(* Offers shapes for a structuring element. *)
	{attribute 'TcIecLibraryType'}
{attribute 'Namespace' := 'Tc3_Vision'}
TYPE ETcVnStructuringElementShape : (
	TCVN_SES_RECTANGLE:=0, 	(* Rectangle *)
	TCVN_SES_CROSS:=1, 	(* Cross *)
	TCVN_SES_ELLIPSE:=2	(* Ellipse *)
) DINT;
END_TYPE

// Data Types/Enumerations/ETcVnTemplateMatchMethod

(* Offes methods for template matching. *)
	{attribute 'TcIecLibraryType'}
{attribute 'Namespace' := 'Tc3_Vision'}
TYPE ETcVnTemplateMatchMethod : (
	TCVN_TMM_SQDIFF:=0, 	(* Squared difference (supports template mask) *)
	TCVN_TMM_SQDIFF_NORMED:=1, 	(* Normalized squared difference *)
	TCVN_TMM_CCORR:=2, 	(* Cross-correlation *)
	TCVN_TMM_CCORR_NORMED:=3, 	(* Normalized cross-correlation (supports template mask) *)
	TCVN_TMM_CCOEFF:=4, 	(* Correlation coefficient *)
	TCVN_TMM_CCOEFF_NORMED:=5	(* Normalized correlation coefficient *)
) DINT;
END_TYPE

// Data Types/Enumerations/ETcVnThresholdType

(* Offers threshold types. *)
	{attribute 'TcIecLibraryType'}
{attribute 'Namespace' := 'Tc3_Vision'}
TYPE ETcVnThresholdType : (
	TCVN_TT_BINARY:=0, 	(* Binary threshold *)
	TCVN_TT_BINARY_INV:=1, 	(* Inverted binary threshold *)
	TCVN_TT_TRUNC:=2, 	(* Truncated threshold (pixels > thresh are set to thresh, others keep their value) *)
	TCVN_TT_TOZERO:=3, 	(* To zero threshold (pixels < thresh are set to zero, others keep their value) *)
	TCVN_TT_TOZERO_INV:=4, 	(* Inverted to zero threshold (pixels > thresh are set to zero, others keep their value) *)
	TCVN_TT_OTSU_BINARY:=8, 	(* Binary threshold with the threshold value selected according to the Otsu algorithm *)
	TCVN_TT_OTSU_BINARY_INV:=9, 	(* Inverted binary threshold with the threshold value selected according to the Otsu algorithm *)
	TCVN_TT_OTSU_TRUNC:=10, 	(* Truncated threshold with the threshold value selected according to the Otsu algorithm *)
	TCVN_TT_OTSU_TOZERO:=11, 	(* To zero threshold with the threshold value selected according to the Otsu algorithm *)
	TCVN_TT_OTSU_TOZERO_INV:=12, 	(* Inverted to zero threshold with the threshold value selected according to the Otsu algorithm *)
	TCVN_TT_TRIANGLE_BINARY:=16, 	(* Binary threshold with the threshold value selected according to the Triangle algorithm *)
	TCVN_TT_TRIANGLE_BINARY_INV:=17, 	(* Inverted binary threshold with the threshold value selected according to the Triangle algorithm *)
	TCVN_TT_TRIANGLE_TRUNC:=18, 	(* Truncated threshold with the threshold value selected according to the Triangle algorithm *)
	TCVN_TT_TRIANGLE_TOZERO:=19, 	(* To zero threshold with the threshold value selected according to the Triangle algorithm *)
	TCVN_TT_TRIANGLE_TOZERO_INV:=20	(* Inverted to zero threshold with the threshold value selected according to the Triangle algorithm *)
) DINT;
END_TYPE

// Data Types/Enumerations/ETcVnVectorCompareMethod

(* Offers methods for vector comparison. *)
	{attribute 'TcIecLibraryType'}
{attribute 'Namespace' := 'Tc3_Vision'}
TYPE ETcVnVectorCompareMethod : (
	TCVN_VCM_EUCLIDEAN:=0, 	(* Euclidean *)
	TCVN_VCM_ELEMENTWISE:=1	(* Elementwise *)
) DINT;
END_TYPE

// Data Types/Enumerations/ETcVnKeypointDetectionTypeAGAST

(* Offers different neighborhood types for AGAST method (For details see paper: E. Mair et al.: Adaptive and Generic Corner Detection Based on the Accelerated Segment Test, 2010). *)
	{attribute 'TcIecLibraryType'}
{attribute 'Namespace' := 'Tc3_Vision'}
TYPE ETcVnKeypointDetectionTypeAGAST : (
	TCVN_KDT_AGAST_5_8:=0, 	(* 5 of 8 *)
	TCVN_KDT_AGAST_7_12d:=1, 	(* 7 of 12 diamond *)
	TCVN_KDT_AGAST_7_12s:=2, 	(* 7 of 12 square *)
	TCVN_KDT_AGAST_9_16:=3	(* 9 of 16 *)
) DINT;
END_TYPE

// Data Types/Enumerations/ETcVnKeypointDetectionTypeFAST

(* Offers different neighborhood types for FAST method (For details see paper: E. Rosten: Machine Learning for High-speed Corner Detection, 2006). *)
	{attribute 'TcIecLibraryType'}
{attribute 'Namespace' := 'Tc3_Vision'}
TYPE ETcVnKeypointDetectionTypeFAST : (
	TCVN_KDT_FAST_5_8:=0, 	(* 5 of 8 *)
	TCVN_KDT_FAST_7_12:=1, 	(* 7 of 12 *)
	TCVN_KDT_FAST_9_16:=2	(* 9 of 16 *)
) DINT;
END_TYPE

// Data Types/Structs/TcVnParamsAGAST

(* Offers parameters for AGAST method. *)
	{attribute 'TcIecLibraryType'}
{attribute 'Namespace' := 'Tc3_Vision'}
TYPE TcVnParamsAGAST : 
	STRUCT
		(* Threshold for the intensity difference between the center pixel and its surrounding circle *)
		nThreshold : DINT := 10;
		(* If true, non-maximum suppression is applied. *)
		bNonMaxSuppression : BOOL := TRUE;
		 {attribute 'hide'}
		_reserved1 : ARRAY [1..3] OF USINT;
		(* Neighborhood type *)
		 {attribute 'GUID' := 'FA6F5C56-A2E3-4BCD-8022-41680719FF8A'}
		 {attribute 'Namespace' := 'Tc3_Vision'}
		eType : ETcVnKeypointDetectionTypeAGAST := TCVN_KDT_AGAST_9_16;
	END_STRUCT
END_TYPE

// Data Types/Structs/TcVnParamsAKAZE

(* Offers parameters for AKAZE method. *)
	{attribute 'TcIecLibraryType'}
{attribute 'Namespace' := 'Tc3_Vision'}
TYPE TcVnParamsAKAZE : 
	STRUCT
		(* Type of the descriptor *)
		 {attribute 'GUID' := 'EFB57555-E4E6-46A8-8672-7CE1494D9FAA'}
		 {attribute 'Namespace' := 'Tc3_Vision'}
		eDescrType : ETcVnFeatureDescriptorTypeAKAZE := TCVN_FDT_AKAZE_MLDB;
		(* Size of the descriptor in bits (only for MLDB; 0 = full size) *)
		nDescrSize : UDINT := 0;
		(* Number of descriptor channels (currently only 3 supported for MLDB) *)
		nDescrChannels : UDINT := 3;
		(* Detector response threshold *)
		fThreshold : REAL := 0.001;
		(* Maximum octave evolution *)
		nOctaves : UDINT := 2;
		(* Number of sublevels per scale level *)
		nOctaveLayers : UDINT := 1;
		(* Diffusivity type *)
		 {attribute 'GUID' := '808733BC-B2E0-4793-A0CE-2F414F4C0F1D'}
		 {attribute 'Namespace' := 'Tc3_Vision'}
		eDiffusivity : ETcVnDiffusivityTypeKAZE := TCVN_DT1_KAZE_PM_G2;
	END_STRUCT
END_TYPE

// Data Types/Structs/TcVnParamsBlobDetection

(* Offers parameters for blob detection *)
	{attribute 'TcIecLibraryType'}
{attribute 'Namespace' := 'Tc3_Vision'}
TYPE TcVnParamsBlobDetection : 
	STRUCT
		(* Enable filtering by area (fMinArea <= area <= fMaxArea); strongly recommended to activate for filtering noise with fMinArea. *)
		bFilterByArea : BOOL := TRUE;
		(* Enable filtering by circularity (fMinCircularity <= circularity(4pi * area / perimeter^2) <= fMaxCircularity). *)
		bFilterByCircularity : BOOL := FALSE;
		(* Enable filtering by convexity (fMinConvexity <= convexity(area / hullArea) <= fMaxConvexity). *)
		bFilterByConvexity : BOOL := FALSE;
		(* Enable filtering by eccentricity (fMinEccentricity <= eccentricity <= fMaxEccentricity). *)
		bFilterByEccentricity : BOOL := FALSE;
		(* Enable filtering by inertia ratio (fMinInertiaRatio <= inertia ratio <= fMaxInertiaRatio). *)
		bFilterByInertiaRatio : BOOL := FALSE;
		 {attribute 'hide'}
		_reserved1 : ARRAY [1..3] OF USINT;
		(* Min estimated blob area in pixel *)
		fMinArea : REAL := 10;
		(* Max estimated blob area in pixel *)
		fMaxArea : REAL := 100000000;
		(* Min circularity (1.0: ideal circle, < 1: less circular, 0: not circular at all) *)
		fMinCircularity : REAL := 0;
		(* Max circularity (1.0: ideal circle, < 1: less circular, 0: not circular at all) *)
		fMaxCircularity : REAL := 1;
		(* Min convexity (1.0: blob fully convex, < 1: less convex) *)
		fMinConvexity : REAL := 0;
		(* Max convexity (1.0: blob fully convex, < 1: less convex) *)
		fMaxConvexity : REAL := 1;
		(* Min eccentricity (0.0: circular, 1.0: linear) *)
		fMinEccentricity : REAL := 0;
		(* Max eccentricity (0.0: circular, 1.0: linear) *)
		fMaxEccentricity : REAL := 1;
		(* Min inertia ratio (1.0: equal width and height, 0.0: linear) *)
		fMinInertiaRatio : REAL := 0;
		(* Max inertia ratio (1.0: equal width and height, 0.0: linear) *)
		fMaxInertiaRatio : REAL := 1;
		(* Threshold type for internally applied threshold method (OTSU_XXX only supported for USINT images). *)
		 {attribute 'GUID' := 'C40D9A7B-C720-49F8-A5B9-1663BB6925B6'}
		 {attribute 'Namespace' := 'Tc3_Vision'}
		eThresholdType : ETcVnThresholdType := TCVN_TT_BINARY;
		(* Threshold to start with (if fThresholdStep > 0, otherwise this is the only threshold used). *)
		fMinThreshold : REAL := 30;
		(* Threshold to end with (if fThresholdStep > 0, otherwise this value is not used). *)
		fMaxThreshold : REAL := 225;
		(* Sets to 0 if only 1 threshold should be used (much faster than multiple thresholds and combining the results). *)
		fThresholdStep : REAL := 0;
		(* Minimum distance between the center points of two different blobs (only used if fThresholdStep > 0; if distance < fMinBlobDistance, the blobs are treated as the same). *)
		fMinBlobDistance : REAL := 5;
		(* Minimum number of threshold steps, for which the same contour has to be detected (only used if fThresholdStep > 0; same means center point distance < fMinBlobDistance). *)
		nMinRepeatability : UDINT := 2;
		(* Selects, which of the multi-threshold blob contours should be returned. *)
		 {attribute 'GUID' := '6B3EA399-FB72-4A3D-A347-965F9D388EB6'}
		 {attribute 'Namespace' := 'Tc3_Vision'}
		eBlobCombination : ETcVnBlobCombination := TCVN_BC_MEDIAN_THRESHOLD;
	END_STRUCT
END_TYPE

// Data Types/Structs/TcVnParamsBRISK

(* Offers parameters for BRISK method. *)
	{attribute 'TcIecLibraryType'}
{attribute 'Namespace' := 'Tc3_Vision'}
TYPE TcVnParamsBRISK : 
	STRUCT
		(* Detection threshold *)
		nThreshold : DINT := 30;
		(* Detection octaves (0 for single scale) *)
		nOctaves : UDINT := 3;
		(* Scale factor for the neighborhood pattern *)
		fPatternScale : REAL := 1;
	END_STRUCT
END_TYPE

// Data Types/Structs/TcVnParamsFAST

(* Offers parameters for FAST method. *)
	{attribute 'TcIecLibraryType'}
{attribute 'Namespace' := 'Tc3_Vision'}
TYPE TcVnParamsFAST : 
	STRUCT
		(* Threshold for the intensity difference between the center pixel and its surrounding circle *)
		nThreshold : DINT := 10;
		(* If true, non-maximum suppression is applied. *)
		bNonMaxSuppression : BOOL := TRUE;
		 {attribute 'hide'}
		_reserved1 : ARRAY [1..3] OF USINT;
		(* Neighborhood type *)
		 {attribute 'GUID' := 'FBD32F44-42B6-42E8-8896-D6A6C0F64387'}
		 {attribute 'Namespace' := 'Tc3_Vision'}
		eType : ETcVnKeypointDetectionTypeFAST := TCVN_KDT_FAST_9_16;
	END_STRUCT
END_TYPE

// Data Types/Structs/TcVnParamsGFTT

(* Offers parameters for GFTT method. *)
	{attribute 'TcIecLibraryType'}
{attribute 'Namespace' := 'Tc3_Vision'}
TYPE TcVnParamsGFTT : 
	STRUCT
		(* Maximum number of corners to return (strongest ones) *)
		nMaxCorners : UDINT := 1000;
		 {attribute 'hide'}
		_reserved1 : UDINT;
		(* Minimum accepted corner quality, relative to the strongest one *)
		fQualityLevel : LREAL := 0.01;
		(* Minimum euclidean distance between returned keypoints *)
		fMinDistance : LREAL := 1;
		(* Neighborhood block size *)
		nBlockSize : UDINT := 3;
		(* If true, a Harris detector is used instead of the default method. *)
		bUseHarrisDetector : BOOL := FALSE;
		 {attribute 'hide'}
		_reserved2 : ARRAY [1..3] OF USINT;
		(* Free parameter of the Harris detector *)
		fHarrisK : LREAL := 0.04;
	END_STRUCT
END_TYPE

// Data Types/Structs/TcVnParamsKAZE

(* Offers parameters for KAZE method *)
	{attribute 'TcIecLibraryType'}
{attribute 'Namespace' := 'Tc3_Vision'}
TYPE TcVnParamsKAZE : 
	STRUCT
		(* If true, the descriptor size is extended from the default 64 byte to 128 byte. *)
		bExtended : BOOL := FALSE;
		(* If true, upright (rotation dependent) descriptors are computed. *)
		bUpright : BOOL := FALSE;
		 {attribute 'hide'}
		_reserved1 : UINT;
		(* Detector response threshold *)
		fThreshold : REAL := 0.001;
		(* Maximum octave evolution of the image *)
		nOctaves : UDINT := 4;
		(* Number of sublevels per scale level *)
		nOctaveLayers : UDINT := 2;
		(* Diffusivity type *)
		 {attribute 'GUID' := '808733BC-B2E0-4793-A0CE-2F414F4C0F1D'}
		 {attribute 'Namespace' := 'Tc3_Vision'}
		eDiffusivity : ETcVnDiffusivityTypeKAZE := TCVN_DT1_KAZE_PM_G2;
	END_STRUCT
END_TYPE

// Data Types/Structs/TcVnParamsMSER

(* Offers parameters for MSER method *)
	{attribute 'TcIecLibraryType'}
{attribute 'Namespace' := 'Tc3_Vision'}
TYPE TcVnParamsMSER : 
	STRUCT
		(* Delta for size comparison *)
		nDelta : DINT := 5;
		(* Minimum blob size *)
		nMinArea : UDINT := 60;
		(* Maximum blob size *)
		nMaxArea : UDINT := 14400;
		 {attribute 'hide'}
		_reserved1 : UDINT;
		(* Maximum blob size variation *)
		fMaxVariation : LREAL := 0.25;
		(* Minimum MSER diversity *)
		fMinDiversity : LREAL := 0.2;
		(* Maximum evolution steps (only used for color images) *)
		nMaxEvolution : UDINT := 200;
		 {attribute 'hide'}
		_reserved2 : UDINT;
		(* Area threshold to cause re-initialization (only used for color images) *)
		fAreaThreshold : LREAL := 1.01;
		(* Minimum margin (only used for color images) *)
		fMinMargin : LREAL := 0.003;
		(* Aperture size for edge bluring (only used for color images) *)
		nEdgeBlurSize : UDINT := 5;
		 {attribute 'hide'}
		_reserved3 : UDINT;
	END_STRUCT
END_TYPE

// Data Types/Structs/TcVnParamsORB

(* Offers parameters for ORB method. *)
	{attribute 'TcIecLibraryType'}
{attribute 'Namespace' := 'Tc3_Vision'}
TYPE TcVnParamsORB : 
	STRUCT
		(* Maximum number of returned keypoints *)
		nMaxPoints : UDINT := 500;
		(* Pyramid decimation ratio (must be greater than 1, should be smaller than 2) *)
		fPyramidScale : REAL := 1.2;
		(* Number of pyramid levels *)
		nPyramidLevels : UDINT := 8;
		(* Size of the border, where no features are detected (should match nPatchSize) *)
		nEdgeThreshold : UDINT := 31;
		(* First pyramid level (currently, only 0 is supported) *)
		nFirstLevel : UDINT := 0;
		(* Number of points to produce each BRIEF descriptor element (2, 3, 4) *)
		nBriefPoints : UDINT := 2;
		(* Score type (HARRIS is more stable but slightly slower than FAST) *)
		 {attribute 'GUID' := '688ACEF5-9A4A-4447-9B39-CBC4558C02DB'}
		 {attribute 'Namespace' := 'Tc3_Vision'}
		eScoreType : ETcVnFeatureScoreTypeORB := TCVN_FST_ORB_HARRIS;
		(* Patch size of the BRIEF descriptor *)
		nPatchSize : UDINT := 31;
		(* Threshold for the FAST keypoint detection *)
		nFastThreshold : DINT := 20;
	END_STRUCT
END_TYPE

// Data Types/Structs/TcVnParamsSB

(* Offers parameters for SB method (a simple blob detector with multiple thresholds). *)
	{attribute 'TcIecLibraryType'}
{attribute 'Namespace' := 'Tc3_Vision'}
TYPE TcVnParamsSB : 
	STRUCT
		(* Enable filtering by area (fMinArea <= area < fMaxArea). *)
		bFilterByArea : BOOL := TRUE;
		(* Enable filtering by circularity (fMinCircularity <= circularity(4pi * area / perimeter^2) < fMaxCircularity). *)
		bFilterByCircularity : BOOL := FALSE;
		(* Enable filtering by color (thresholdedColor(0 or 255) = nBlobColor). *)
		bFilterByColor : BOOL := FALSE;
		(* Enable filtering by convexity (fMinConvexity <= convexity(area / hullArea) < fMaxConvexity). *)
		bFilterByConvexity : BOOL := FALSE;
		(* Enable filtering by inertia ratio (fMinInertiaRatio <= inertia ratio < fMaxInertiaRatio). *)
		bFilterByInertia : BOOL := FALSE;
		 {attribute 'hide'}
		_reserved1 : ARRAY [1..3] OF USINT;
		(* Min estimated blob area in pixel *)
		fMinArea : REAL := 25;
		(* Max estimated blob area in pixel *)
		fMaxArea : REAL := 15000;
		(* Min circularity (1.0: ideal circle, < 1: less circular, 0: not circular at all) *)
		fMinCircularity : REAL := 0;
		(* Max circularity (1.0: ideal circle, < 1: less circular, 0: not circular at all) *)
		fMaxCircularity : REAL := 1;
		(* 0 or 255 *)
		nBlobColor : USINT := 255;
		 {attribute 'hide'}
		_reserved2 : ARRAY [1..3] OF USINT;
		(* Min convexity (1.0: blob fully convex, < 1: less convex) *)
		fMinConvexity : REAL := 0;
		(* Max convexity (1.0: blob fully convex, < 1: less convex) *)
		fMaxConvexity : REAL := 1;
		(* Min inertia ratio (0.0 .. 1.0) *)
		fMinInertiaRatio : REAL := 0;
		(* Max inertia ratio (0.0 .. 1.0) *)
		fMaxInertiaRatio : REAL := 1;
		(* Min distance between different blobs *)
		fMinBlobDist : REAL := 5;
		(* Min number of same detected blobs (dist < fMinBlobDist) in different thresholds *)
		nMinRepeatability : UDINT := 2;
		(* Min threshold (start) *)
		fMinThreshold : REAL := 30;
		(* Max threshold (stop) *)
		fMaxThreshold : REAL := 225;
		(* Threshold step between min and max threshold *)
		fThresholdStep : REAL := 10;
	END_STRUCT
END_TYPE

// Version/Global_Version
{attribute 'TcGenerated'}
// This function has been automatically generated from the project information.
VAR_GLOBAL CONSTANT
	{attribute 'const_non_replaced'}
	{attribute 'linkalways'}
	stLibVersion_Tc3_Vision : ST_LibVersion := (iMajor := 4, iMinor := 0, iBuild := 2, iRevision := 13, sVersion := '4.0.2.13');
	{attribute 'const_non_replaced'}
	{attribute 'linkalways'}
	sLibraryId_Tc3_Vision : String := 'Beckhoff Automation GmbH|Tc3_Vision|4.0.2.13';
END_VAR

// Global Variables/Global_Variables

	VAR_GLOBAL
		VISION_ADS_TIMEOUT	:	TIME := TIME#5s;	(* Default ADS timeout. *)
	END_VAR

// Global Variables/TC3_VISION_IID_LIST

	VAR_GLOBAL
		IID_ITcVnColorModel	:	IID := (Data1 := 16#AFF801F3, Data2 := 16#60D0, Data3 := 16#43FA, Data4 := [16#98, 16#0F, 16#57, 16#2A, 16#62, 16#05, 16#B5, 16#AF]);	(* Interface ID for interface ITcVnColorModel *)
	END_VAR

// Function Blocks/Image Acquisition/FB_VN_GevCameraControl

	{attribute 'c++_compatible'}
	{attribute 'external_name' := 'FB_VN_GevCameraControl_GUID_B1A3978C_F082_3A85_2169_138C29DFB3DA'}
	{attribute 'TcIecLibraryType'}
	{attribute 'no_explicit_call' :='do not call this POU directly'}
	(* This FB provides the basic functionality to control a GigE Vision camera and access its calibration data. *)
	FUNCTION_BLOCK FB_VN_GevCameraControl
	VAR
		(* Internal reference to the corresponding TcVnGevImageProvider TcCOM module ID, which needs to be set via TC init symbol. *)
		{attribute 'TcInitSymbol'}
		{attribute 'TcCategoryOID' := 'TcVnGevImageProvider'}
		 {attribute 'GUID' := '18071995-0000-0000-0000-00000000000F'}
		oidITcVnGevImageProvider : OTCID;
		 {attribute 'hide'}
		_reserved1 : UINT_0_32;
		(* Internal stuff *)
		{attribute 'hide'}
		 {attribute 'GUID' := '18071995-0000-0000-0000-000000000018'}
		pInternal : PVOID;
	END_VAR


	(* Delete all images contained in the TcVnGevImageProvider TcCOM module receive queue and reset the corresponding omitted images counter. *)
	METHOD ClearImageQueue : HRESULT
END_METHOD


	(* Close the control channel to the camera. *)
	METHOD CloseCamera : HRESULT
END_METHOD


	(* Internal method *)
	{attribute 'hide'}
	METHOD FB_exit : BOOL
	VAR_INPUT
		(*  if TRUE, the exit method is called for exiting an instance that is copied afterwards (online change). *)
		bInCopyCode : BOOL;
	END_VAR
END_METHOD


	(* Internal method *)
	{attribute 'hide'}
	METHOD FB_init : BOOL
	VAR_INPUT
		(*  if TRUE, the retain variables are initialized (warm start / cold start) *)
		bInitRetains : BOOL;
		(*  if TRUE, the instance afterwards gets moved into the copy code (online change) *)
		bInCopyCode : BOOL;
	END_VAR
END_METHOD


	(* Gets the reference calibration pattern points from the TcVnGevImageProvider TcCOM module (Can be set from the calibration assistant) *)
	METHOD GetCalibPatternRef : HRESULT
	VAR_INPUT
		(* Returns the reference calibration pattern points (ContainerType_Vector_TcVnPoint3_REAL) *)
 {attribute 'GUID' := 'BC72B333-E095-465B-9693-7979773CA3B8'}
				ipCalibPatternRef : REFERENCE TO ITcVnContainer;
	END_VAR
END_METHOD


	(* Gets the camera matrix from the TcVnGevImageProvider TcCOM module (requires intrinsic calibration parameters, e.g. set by the calibration assistant) *)
	METHOD GetCameraMatrix : HRESULT
	VAR_INPUT
		(* Returns the camera matrix *)
 {attribute 'GUID' := '91A420A3-4727-4481-B3BB-170528E5BC7C'}
		 {attribute 'Namespace' := 'VN'}
				aCameraMatrix : REFERENCE TO TcVnMatrix3x3_LREAL;
	END_VAR
END_METHOD


	(* Gets the current available image (first in receive queue). *)
	METHOD GetCurrentImage : HRESULT
	VAR_INPUT
		(* Returns the image *)
 {attribute 'GUID' := '70D42C6D-6F4E-4719-8B29-2883D5D59B1C'}
				ipImage : REFERENCE TO ITcVnImage;
	END_VAR
END_METHOD


	(* Gets the current available image (first in receive queue) with undistortion applied (requires intrinsic calibration parameters in the TcVnGevImageProvider TcCOM module, e.g. set by the calibration assistant) *)
	METHOD GetCurrentImageUndistorted : HRESULT
	VAR_INPUT
		(* Returns the undistorted image *)
 {attribute 'GUID' := '70D42C6D-6F4E-4719-8B29-2883D5D59B1C'}
				ipImage : REFERENCE TO ITcVnImage;
	END_VAR
END_METHOD


	(* Gets the current available image (first in receive queue) and its corresponding GVSP info. *)
	METHOD GetCurrentImageWithGvspInfo : HRESULT
	VAR_INPUT
		(* Returns the image *)
 {attribute 'GUID' := '70D42C6D-6F4E-4719-8B29-2883D5D59B1C'}
				ipImage : REFERENCE TO ITcVnImage;
		(* Returns the GVSP info *)
 {attribute 'GUID' := '63FC7E33-91CD-44CD-9015-0BD1DC25722C'}
				stGvspInfo : REFERENCE TO GVSP_IMAGE_INFO;
	END_VAR
END_METHOD


	(* Gets the current available image (first in receive queue) with its corresponding GVSP info and undistortion applied (requires intrinsic calibration parameters in the TcVnGevImageProvider TcCOM module, e.g. set by the calibration assistant) *)
	METHOD GetCurrentImageWithGvspInfoUndistorted : HRESULT
	VAR_INPUT
		(* Returns the undistorted image *)
 {attribute 'GUID' := '70D42C6D-6F4E-4719-8B29-2883D5D59B1C'}
				ipImage : REFERENCE TO ITcVnImage;
		(* Returns the GVSP info *)
 {attribute 'GUID' := '63FC7E33-91CD-44CD-9015-0BD1DC25722C'}
				stGvspInfo : REFERENCE TO GVSP_IMAGE_INFO;
	END_VAR
END_METHOD


	(* Gets the distortion coefficients from the TcVnGevImageProvider TcCOM module (requires intrinsic calibration parameters, e.g. set by the calibration assistant) *)
	METHOD GetDistortionCoefficients : HRESULT
	VAR_INPUT
		(* Returns the distortion coefficients [k1, k2, p1, p2, k3, k4, k5, k6] *)
 {attribute 'GUID' := 'DD112102-C23A-4B37-A43A-A96400B57010'}
		 {attribute 'Namespace' := 'VN'}
				aDistortionCoefficients : REFERENCE TO TcVnArray8_LREAL;
	END_VAR
END_METHOD


	(* Gets the last received image from the queue. *)
	METHOD GetLastImageFromQueue : HRESULT
	VAR_INPUT
		(* Returns the image *)
 {attribute 'GUID' := '70D42C6D-6F4E-4719-8B29-2883D5D59B1C'}
				ipImage : REFERENCE TO ITcVnImage;
	END_VAR
END_METHOD


	(* Gets the number of omitted images since the last call of ClearImageQueue(). If the image receive queue in the TcVnGevImageProvider TcCOM module is full and a new image arrives, the first one in the queue will be deleted and the omitted counter is increased. *)
	METHOD GetOmittedImagesNum : HRESULT
	VAR_INPUT
		(* Returns the number of omitted images *)
		nOmitted : REFERENCE TO ULINT;
	END_VAR
END_METHOD


	(* Gets the rotation matrix from the TcVnGevImageProvider TcCOM module (requires extrinsic calibration parameters, e.g. set by the calibration assistant) *)
	METHOD GetRotationMatrix : HRESULT
	VAR_INPUT
		(* Returns the rotation matrix *)
 {attribute 'GUID' := '91A420A3-4727-4481-B3BB-170528E5BC7C'}
		 {attribute 'Namespace' := 'VN'}
				aRotationMatrix : REFERENCE TO TcVnMatrix3x3_LREAL;
	END_VAR
END_METHOD


	(* Gets the current state of the internal camera control state machine. *)
	METHOD GetState : ETcVnCameraState
END_METHOD


	(* Gets the translation vector from the TcVnGevImageProvider TcCOM module (requires extrinsic calibration parameters, e.g. set by the calibration assistant) *)
	METHOD GetTranslationVector : HRESULT
	VAR_INPUT
		(* Returns the translation vector *)
 {attribute 'GUID' := 'B9A67DEB-A7D1-4F25-95A3-4A82FA5C1E28'}
		 {attribute 'Namespace' := 'VN'}
				aTranslationVector : REFERENCE TO TcVnVector3_LREAL;
	END_VAR
END_METHOD


	(* Initialize the camera to the intended state (includes sending the 'InitCameraCommands' defined in the GevImageAcquisition TcCOM module to the camera). *)
	METHOD InitializeCamera : HRESULT
END_METHOD


	(* Open a control channel to the camera. *)
	METHOD OpenCamera : HRESULT
END_METHOD


	(* Reset the camera controller to initial state (might require multiple calls depending on current state, until S_OK is returned) *)
	METHOD Reset : HRESULT
END_METHOD


	(* Reset the camera features to initial state (sends the 'InitCameraCommands' defined in the GevImageAcquisition TcCOM module to the camera). *)
	METHOD ResetCameraFeatures : HRESULT
END_METHOD


	(* Sets the camera matrix to the TcVnGevImageProvider TcCOM module *)
	METHOD SetCameraMatrix : HRESULT
	VAR_INPUT
		(* The camera matrix to be copied to the TcCOM module *)
 {attribute 'GUID' := '91A420A3-4727-4481-B3BB-170528E5BC7C'}
		 {attribute 'Namespace' := 'VN'}
				aCameraMatrix : REFERENCE TO TcVnMatrix3x3_LREAL;
	END_VAR
END_METHOD


	(* Sets the distortion coefficients to the TcVnGevImageProvider TcCOM module *)
	METHOD SetDistortionCoefficients : HRESULT
	VAR_INPUT
		(* The distortion coefficients to be copied to the TcCOM module *)
 {attribute 'GUID' := 'DD112102-C23A-4B37-A43A-A96400B57010'}
		 {attribute 'Namespace' := 'VN'}
				aDistortionCoefficients : REFERENCE TO TcVnArray8_LREAL;
	END_VAR
END_METHOD


	(* Sets the rotation matrix to the TcVnGevImageProvider TcCOM module *)
	METHOD SetRotationMatrix : HRESULT
	VAR_INPUT
		(* The rotation matrix to be copied to the TcCOM module *)
 {attribute 'GUID' := '91A420A3-4727-4481-B3BB-170528E5BC7C'}
		 {attribute 'Namespace' := 'VN'}
				aRotationMatrix : REFERENCE TO TcVnMatrix3x3_LREAL;
	END_VAR
END_METHOD


	(* Sets the translation vector to the TcVnGevImageProvider TcCOM module *)
	METHOD SetTranslationVector : HRESULT
	VAR_INPUT
		(* The translation vector to be copied to the TcCOM module *)
 {attribute 'GUID' := 'B9A67DEB-A7D1-4F25-95A3-4A82FA5C1E28'}
		 {attribute 'Namespace' := 'VN'}
				aTranslationVector : REFERENCE TO TcVnVector3_LREAL;
	END_VAR
END_METHOD


	(* Send the 'StartAcquisitionCommands' defined in the TcVnGevImageProvider TcCOM module to the camera. *)
	METHOD StartAcquisition : HRESULT
END_METHOD


	(* Send the 'StopAcquisitionCommands' defined in the TcVnGevImageProvider TcCOM module to the camera. *)
	METHOD StopAcquisition : HRESULT
END_METHOD


	(* Send the 'SoftwareTriggerCommands' defined in the TcVnGevImageProvider TcCOM module to the camera. *)
	METHOD TriggerImage : HRESULT
END_METHOD

END_FUNCTION_BLOCK

// Function Blocks/Image Acquisition/FB_VN_FileSourceControl

	{attribute 'c++_compatible'}
	{attribute 'external_name' := 'FB_VN_FileSourceControl_GUID_4F53D607_3B4C_364C_3211_1EEDF57CF9AE'}
	{attribute 'TcIecLibraryType'}
	{attribute 'no_explicit_call' :='do not call this POU directly'}
	(* This FB provides access to the images send by a File Source instance. *)
	FUNCTION_BLOCK FB_VN_FileSourceControl
	VAR
		(* Internal reference to the corresponding TcVnFileImageProvider TcCOM module ID, which needs to be set via TC init symbol. *)
		{attribute 'TcInitSymbol'}
		{attribute 'TcCategoryOID' := 'TcVnFileImageProvider'}
		 {attribute 'GUID' := '18071995-0000-0000-0000-00000000000F'}
		oidITcVnFileImageProvider : OTCID;
		 {attribute 'hide'}
		_reserved1 : UINT_0_32;
		(* Internal reference to private data. *)
		{attribute 'hide'}
		 {attribute 'GUID' := '18071995-0000-0000-0000-000000000018'}
		pPriv : PVOID;
	END_VAR


	(* Internal method *)
	{attribute 'hide'}
	METHOD FB_exit : BOOL
	VAR_INPUT
		(* If TRUE, the exit method is called for exiting an instance that is copied afterwards (online change). *)
		bInCopyCode : BOOL;
	END_VAR
END_METHOD


	(* Internal method *)
	{attribute 'hide'}
	METHOD FB_init : BOOL
	VAR_INPUT
		(* If TRUE, the retain variables are initialized (warm start / cold start) *)
		bInitRetains : BOOL;
		(* If TRUE, the exit method is called for exiting an instance that is copied afterwards (online change). *)
		bInCopyCode : BOOL;
	END_VAR
END_METHOD


	(* Gets the current available image (if any). *)
	METHOD GetCurrentImage : HRESULT
	VAR_INPUT
		(* Returns the image *)
 {attribute 'GUID' := '70D42C6D-6F4E-4719-8B29-2883D5D59B1C'}
				ipImage : REFERENCE TO ITcVnImage;
	END_VAR
END_METHOD


	(* Gets the current available image (if any) and the corresponding file name. *)
	METHOD GetCurrentImageAndFileName : HRESULT
	VAR_INPUT
		(* Returns the image *)
 {attribute 'GUID' := '70D42C6D-6F4E-4719-8B29-2883D5D59B1C'}
				ipImage : REFERENCE TO ITcVnImage;
	END_VAR
	VAR_IN_OUT CONSTANT
		(* Returns the file name *)
 {attribute 'GUID' := '18071995-0000-0000-0000-00000000001A'}
				sFileName : STRING;
	END_VAR
	VAR_INPUT
		(* Define the maximum allowed length for the file name *)
		nMaxLen : UINT;
	END_VAR
END_METHOD


	(* Activates the File Source. If not in trigger mode, it will start sending images. *)
	METHOD StartAcquisition : HRESULT
END_METHOD


	(* Deactivates the File Source. It will stop sending images. *)
	METHOD StopAcquisition : HRESULT
END_METHOD


	(* Reset the controller to initial state (might require multiple calls depending on current state, until S_OK is returned) *)
	METHOD Reset : HRESULT
END_METHOD


	(* Gets the current state of the internal camera control state machine. *)
	METHOD GetState : ETcVnCameraState
END_METHOD


	(* If in trigger mode, this function triggers the next image in the list. *)
	METHOD TriggerImage : HRESULT
END_METHOD


	(* If in trigger mode, this function triggers a specific image in the list. *)
	METHOD TriggerImageExp : HRESULT
	VAR_INPUT
		(* Amount of images to skip, relative to current *)
		nSkipImages : DINT;
	END_VAR
END_METHOD


	(* If in trigger mode, this function triggers a specific image in the list by name. *)
	METHOD TriggerImageByName : HRESULT
	VAR_IN_OUT CONSTANT
		(* Name of the image to trigger *)
 {attribute 'GUID' := '18071995-0000-0000-0000-00000000001A'}
				sImageName : STRING;
	END_VAR
END_METHOD

END_FUNCTION_BLOCK

// Function Blocks/Image Acquisition/FB_VN_SimpleCameraControl

	{attribute 'c++_compatible'}
	{attribute 'external_name' := 'FB_VN_SimpleCameraControl_GUID_C57D481C_6AC1_3CDC_211F_5C11AC3CD922'}
	{attribute 'TcIecLibraryType'}
	{attribute 'no_explicit_call' :='do not call this POU directly'}
	(* This FB provides the basic functionality to control a camera or a FileSource. *)
	FUNCTION_BLOCK FB_VN_SimpleCameraControl
	VAR
		(* Internal reference to the corresponding TcVnImageProvider TcCOM module ID, which needs to be set via TC init symbol. *)
		{attribute 'TcInitSymbol'}
		{attribute 'TcCategoryOID' := 'TcVnImageProvider'}
		 {attribute 'GUID' := '18071995-0000-0000-0000-00000000000F'}
		oidITcVnImageProvider : OTCID;
		 {attribute 'hide'}
		_reserved1 : UINT_0_32;
		(* Internal stuff *)
		{attribute 'hide'}
		 {attribute 'GUID' := '18071995-0000-0000-0000-000000000018'}
		pInternal : PVOID;
	END_VAR


	(* Internal method *)
	{attribute 'hide'}
	METHOD FB_exit : BOOL
	VAR_INPUT
		(*  if TRUE, the exit method is called for exiting an instance that is copied afterwards (online change). *)
		bInCopyCode : BOOL;
	END_VAR
END_METHOD


	(* Internal method *)
	{attribute 'hide'}
	METHOD FB_init : BOOL
	VAR_INPUT
		(*  if TRUE, the retain variables are initialized (warm start / cold start) *)
		bInitRetains : BOOL;
		(*  if TRUE, the instance afterwards gets moved into the copy code (online change) *)
		bInCopyCode : BOOL;
	END_VAR
END_METHOD


	(* Get the current available image (if any). *)
	METHOD GetCurrentImage : HRESULT
	VAR_INPUT
		(* Returns the image *)
 {attribute 'GUID' := '70D42C6D-6F4E-4719-8B29-2883D5D59B1C'}
				ipImage : REFERENCE TO ITcVnImage;
	END_VAR
END_METHOD


	(* Get the current state of the internal camera control state machine. *)
	METHOD GetState : ETcVnCameraState
END_METHOD


	(* Reset the camera to initial state (might require multiple calls depending on current state, until S_OK is returned) *)
	METHOD Reset : HRESULT
END_METHOD


	(* Start the image acquisition. *)
	METHOD StartAcquisition : HRESULT
END_METHOD


	(* Stop the image acquisition. *)
	METHOD StopAcquisition : HRESULT
END_METHOD


	(* Trigger the next image. *)
	METHOD TriggerImage : HRESULT
END_METHOD

END_FUNCTION_BLOCK

// Function Blocks/File Access/FB_VN_ReadCalibrationPattern

	{attribute 'c++_compatible'}
	{attribute 'external_name' := 'FB_VN_ReadCalibrationPattern_GUID_F379CE3F_BDCE_345C_3434_ADFB5334B83F'}
	{attribute 'TcIecLibraryType'}
	(* This FB reads calibration pattern reference points from an xml file on the targte pc. *)
	FUNCTION_BLOCK FB_VN_ReadCalibrationPattern
	VAR_IN_OUT CONSTANT
		(* Full path of the file or relative path to the default directory on the target pc (%TWINCAT3DIR%\\CustomConfig\\Vision\\CalibrationPattern) *)
		 {attribute 'GUID' := '18071995-0000-0000-0000-00000000001A'}
		sFilePath : STRING;
	END_VAR
	VAR_INPUT
		(* Returns a container with the pattern points (ContainerType_Vector_TcVnPoint3_REAL) *)
		 {attribute 'GUID' := 'BC72B333-E095-465B-9693-7979773CA3B8'}
		ipDestContainer : REFERENCE TO ITcVnContainer;
		(* Reading the file is triggered by a rising edge at this input. *)
		bRead : BOOL;
	END_VAR
	VAR
		 {attribute 'hide'}
		_reserved1 : ARRAY [1..3] OF USINT;
	END_VAR
	VAR_INPUT
		(* Indicates the time before the function is cancelled. *)
		nTimeout : TIME := VISION_ADS_TIMEOUT;
	END_VAR
	VAR_OUTPUT
		(* This output remains TRUE until the function block has executed a command, but at the longest for the duration supplied to the 'nTimeout' input. While bBusy = TRUE, no new command will be accepted at the inputs. *)
		bBusy : BOOL;
		(* This output is switched to TRUE as soon as an error occurs during the execution of a command. The command-specific error code is contained in ‘nErrorId’. If the function block has a timeout error, 'bError' is TRUE and 'nErrorId' is 1861 (hexadecimal 0x745). Is reset to FALSE by the execution of a command at the inputs. *)
		bError : BOOL;
	END_VAR
	VAR
		 {attribute 'hide'}
		_reserved2 : UINT;
	END_VAR
	VAR_OUTPUT
		(* Contains the ADS error code or the command-specific error code of the last executed command. Is reset to 0 by the execution of a command at the inputs. *)
		nErrorId : UDINT;
	END_VAR
	VAR
		(* Internal parameter *)
		{attribute 'hide'}
		nAdsInvStamp : UINT;
		(* Internal parameter *)
		{attribute 'hide'}
		nAdsInvCnt : BYTE;
		(* Internal parameter *)
		{attribute 'hide'}
		ePendingRequest : BYTE;
		(* Internal parameter *)
		{attribute 'hide'}
		nTimeElapsed : TIME;
		(* Internal parameter *)
		{attribute 'hide'}
		bLastRead : BOOL;
		 {attribute 'hide'}
		_reserved3 : UINT_24_56;
		(* Internal parameter *)
		{attribute 'hide'}
		 {attribute 'GUID' := '18071995-0000-0000-0000-000000000018'}
		pBuffer : PVOID;
		(* Internal parameter *)
		{attribute 'hide'}
		 {attribute 'GUID' := '18071995-0000-0000-0000-000000000018'}
		pFilePathPending : PVOID;
	END_VAR


	(* Internal method *)
	{attribute 'hide'}
	METHOD FB_exit : BOOL
	VAR_INPUT
		(*  if TRUE, the exit method is called for exiting an instance that is copied afterwards (online change). *)
		bInCopyCode : BOOL;
	END_VAR
END_METHOD


	(* Internal method *)
	{attribute 'hide'}
	METHOD FB_init : BOOL
	VAR_INPUT
		(*  if TRUE, the retain variables are initialized (warm start / cold start) *)
		bInitRetains : BOOL;
		(*  if TRUE, the instance afterwards gets moved into the copy code (online change) *)
		bInCopyCode : BOOL;
	END_VAR
END_METHOD

END_FUNCTION_BLOCK

// Function Blocks/File Access/FB_VN_ReadContainer

	{attribute 'c++_compatible'}
	{attribute 'external_name' := 'FB_VN_ReadContainer_GUID_09A9DCF0_604B_34FA_0D21_93B42780019C'}
	{attribute 'TcIecLibraryType'}
	(* This FB reads a container from an xml file on the target pc. *)
	FUNCTION_BLOCK FB_VN_ReadContainer
	VAR_IN_OUT CONSTANT
		(* Full path of the file or relative path to the default directory on the target pc *)
		 {attribute 'GUID' := '18071995-0000-0000-0000-00000000001A'}
		sFilePath : STRING;
	END_VAR
	VAR_INPUT
		(* Returns a container with the loaded content *)
		 {attribute 'GUID' := 'BC72B333-E095-465B-9693-7979773CA3B8'}
		ipDestContainer : REFERENCE TO ITcVnContainer;
		(* The type id of the container to return. If this parameter is not set, a suitable container type will be determined automatically (except for csv files). *)
		 {attribute 'GUID' := '18071995-0000-0000-0000-000000000021'}
		nDestTypeGuid : GUID;
		(* Reading the file is triggered by a rising edge at this input. *)
		bRead : BOOL;
	END_VAR
	VAR
		 {attribute 'hide'}
		_reserved1 : ARRAY [1..3] OF USINT;
	END_VAR
	VAR_INPUT
		(* Indicates the time before the function is cancelled. *)
		nTimeout : TIME := VISION_ADS_TIMEOUT;
	END_VAR
	VAR_OUTPUT
		(* This output remains TRUE until the function block has executed a command, but at the longest for the duration supplied to the 'nTimeout' input. While bBusy = TRUE, no new command will be accepted at the inputs. *)
		bBusy : BOOL;
		(* This output is switched to TRUE as soon as an error occurs during the execution of a command. The command-specific error code is contained in ‘nErrorId’. If the function block has a timeout error, 'bError' is TRUE and 'nErrorId' is 1861 (hexadecimal 0x745). Is reset to FALSE by the execution of a command at the inputs. *)
		bError : BOOL;
	END_VAR
	VAR
		 {attribute 'hide'}
		_reserved2 : UINT;
	END_VAR
	VAR_OUTPUT
		(* Contains the ADS error code or the command-specific error code of the last executed command. Is reset to 0 by the execution of a command at the inputs. *)
		nErrorId : UDINT;
	END_VAR
	VAR
		(* Internal parameter *)
		{attribute 'hide'}
		nAdsInvStamp : UINT;
		(* Internal parameter *)
		{attribute 'hide'}
		nAdsInvCnt : BYTE;
		(* Internal parameter *)
		{attribute 'hide'}
		ePendingRequest : BYTE;
		(* Internal parameter *)
		{attribute 'hide'}
		nTimeElapsed : TIME;
		(* Internal parameter *)
		{attribute 'hide'}
		bLastRead : BOOL;
		 {attribute 'hide'}
		_reserved3 : UINT_24_56;
		(* Internal parameter *)
		{attribute 'hide'}
		 {attribute 'GUID' := '18071995-0000-0000-0000-000000000018'}
		pReadBuffer : PVOID;
		(* Internal parameter *)
		{attribute 'hide'}
		 {attribute 'GUID' := '18071995-0000-0000-0000-000000000018'}
		pWriteBuffer : PVOID;
		(* Internal parameter *)
		{attribute 'hide'}
		nWriteSize : UDINT;
		 {attribute 'hide'}
		_reserved4 : UINT_0_32;
	END_VAR


	(* Internal method *)
	{attribute 'hide'}
	METHOD FB_exit : BOOL
	VAR_INPUT
		(*  if TRUE, the exit method is called for exiting an instance that is copied afterwards (online change). *)
		bInCopyCode : BOOL;
	END_VAR
END_METHOD


	(* Internal method *)
	{attribute 'hide'}
	METHOD FB_init : BOOL
	VAR_INPUT
		(*  if TRUE, the retain variables are initialized (warm start / cold start) *)
		bInitRetains : BOOL;
		(*  if TRUE, the instance afterwards gets moved into the copy code (online change) *)
		bInCopyCode : BOOL;
	END_VAR
END_METHOD

END_FUNCTION_BLOCK

// Function Blocks/File Access/FB_VN_ReadImage

	{attribute 'c++_compatible'}
	{attribute 'external_name' := 'FB_VN_ReadImage_GUID_9CFBB651_1DA3_3417_10F1_2AF0526B92A7'}
	{attribute 'TcIecLibraryType'}
	(* This FB reads an image from a file on the target pc. *)
	FUNCTION_BLOCK FB_VN_ReadImage
	VAR_IN_OUT CONSTANT
		(* Full path of the file or relative path to the default image directory on the target pc *)
		 {attribute 'GUID' := '18071995-0000-0000-0000-00000000001A'}
		sFilePath : STRING;
	END_VAR
	VAR_INPUT
		(* Returns an image with the loaded content *)
		 {attribute 'GUID' := '70D42C6D-6F4E-4719-8B29-2883D5D59B1C'}
		ipDestImage : REFERENCE TO ITcVnImage;
		(* Reading the file is triggered by a rising edge at this input. *)
		bRead : BOOL;
	END_VAR
	VAR
		 {attribute 'hide'}
		_reserved1 : ARRAY [1..3] OF USINT;
	END_VAR
	VAR_INPUT
		(* Indicates the time before the function is cancelled. *)
		nTimeout : TIME := VISION_ADS_TIMEOUT;
	END_VAR
	VAR_OUTPUT
		(* This output remains TRUE until the function block has executed a command, but at the longest for the duration supplied to the 'nTimeout' input. While bBusy = TRUE, no new command will be accepted at the inputs. *)
		bBusy : BOOL;
		(* This output is switched to TRUE as soon as an error occurs during the execution of a command. The command-specific error code is contained in ‘nErrorId’. If the function block has a timeout error, 'bError' is TRUE and 'nErrorId' is 1861 (hexadecimal 0x745). Is reset to FALSE by the execution of a command at the inputs. *)
		bError : BOOL;
	END_VAR
	VAR
		 {attribute 'hide'}
		_reserved2 : UINT;
	END_VAR
	VAR_OUTPUT
		(* Contains the ADS error code or the command-specific error code of the last executed command. Is reset to 0 by the execution of a command at the inputs. *)
		nErrorId : UDINT;
	END_VAR
	VAR
		(* Internal parameter *)
		{attribute 'hide'}
		nAdsInvStamp : UINT;
		(* Internal parameter *)
		{attribute 'hide'}
		nAdsInvCnt : BYTE;
		(* Internal parameter *)
		{attribute 'hide'}
		ePendingRequest : BYTE;
		(* Internal parameter *)
		{attribute 'hide'}
		nTimeElapsed : TIME;
		(* Internal parameter *)
		{attribute 'hide'}
		bLastRead : BOOL;
		 {attribute 'hide'}
		_reserved3 : UINT_24_56;
		(* Internal parameter *)
		{attribute 'hide'}
		 {attribute 'GUID' := '18071995-0000-0000-0000-000000000018'}
		pBuffer : PVOID;
		(* Internal parameter *)
		{attribute 'hide'}
		 {attribute 'GUID' := '18071995-0000-0000-0000-000000000018'}
		pFilePathPending : PVOID;
	END_VAR


	(* Internal method *)
	{attribute 'hide'}
	METHOD FB_exit : BOOL
	VAR_INPUT
		(*  if TRUE, the exit method is called for exiting an instance that is copied afterwards (online change). *)
		bInCopyCode : BOOL;
	END_VAR
END_METHOD


	(* Internal method *)
	{attribute 'hide'}
	METHOD FB_init : BOOL
	VAR_INPUT
		(*  if TRUE, the retain variables are initialized (warm start / cold start) *)
		bInitRetains : BOOL;
		(*  if TRUE, the instance afterwards gets moved into the copy code (online change) *)
		bInCopyCode : BOOL;
	END_VAR
END_METHOD

END_FUNCTION_BLOCK

// Function Blocks/File Access/FB_VN_ReadMlModel

	{attribute 'c++_compatible'}
	{attribute 'external_name' := 'FB_VN_ReadMlModel_GUID_40256FBA_F075_3791_0CA2_A067683CFCA9'}
	{attribute 'TcIecLibraryType'}
	(* This FB reads a machine learning model from a file on the target pc. *)
	FUNCTION_BLOCK FB_VN_ReadMlModel
	VAR_IN_OUT CONSTANT
		(* Full path of the file or relative path to the default directory on the target pc *)
		 {attribute 'GUID' := '18071995-0000-0000-0000-00000000001A'}
		sFilePath : STRING;
	END_VAR
	VAR_INPUT
		(* Returns the loaded machine learning model *)
		 {attribute 'GUID' := 'AC23D64B-CDFA-4D43-AE8B-364A856EB3E2'}
		ipDestMlModel : REFERENCE TO ITcVnMlModel;
		(* Reading the file is triggered by a rising edge at this input. *)
		bRead : BOOL;
	END_VAR
	VAR
		 {attribute 'hide'}
		_reserved1 : ARRAY [1..3] OF USINT;
	END_VAR
	VAR_INPUT
		(* Indicates the time before the function is cancelled. *)
		nTimeout : TIME := VISION_ADS_TIMEOUT;
	END_VAR
	VAR_OUTPUT
		(* This output remains TRUE until the function block has executed a command, but at the longest for the duration supplied to the 'nTimeout' input. While bBusy = TRUE, no new command will be accepted at the inputs. *)
		bBusy : BOOL;
		(* This output is switched to TRUE as soon as an error occurs during the execution of a command. The command-specific error code is contained in ‘nErrorId’. If the function block has a timeout error, 'bError' is TRUE and 'nErrorId' is 1861 (hexadecimal 0x745). Is reset to FALSE by the execution of a command at the inputs. *)
		bError : BOOL;
	END_VAR
	VAR
		 {attribute 'hide'}
		_reserved2 : UINT;
	END_VAR
	VAR_OUTPUT
		(* Contains the ADS error code or the command-specific error code of the last executed command. Is reset to 0 by the execution of a command at the inputs. *)
		nErrorId : UDINT;
	END_VAR
	VAR
		(* Internal parameter *)
		{attribute 'hide'}
		nAdsInvStamp : UINT;
		(* Internal parameter *)
		{attribute 'hide'}
		nAdsInvCnt : BYTE;
		(* Internal parameter *)
		{attribute 'hide'}
		ePendingRequest : BYTE;
		(* Internal parameter *)
		{attribute 'hide'}
		nTimeElapsed : TIME;
		(* Internal parameter *)
		{attribute 'hide'}
		bLastRead : BOOL;
		 {attribute 'hide'}
		_reserved3 : UINT_24_56;
		(* Internal parameter *)
		{attribute 'hide'}
		 {attribute 'GUID' := '18071995-0000-0000-0000-000000000018'}
		pBuffer : PVOID;
		(* Internal parameter *)
		{attribute 'hide'}
		 {attribute 'GUID' := '18071995-0000-0000-0000-000000000018'}
		pFilePathPending : PVOID;
	END_VAR


	(* Internal method *)
	{attribute 'hide'}
	METHOD FB_exit : BOOL
	VAR_INPUT
		(*  if TRUE, the exit method is called for exiting an instance that is copied afterwards (online change). *)
		bInCopyCode : BOOL;
	END_VAR
END_METHOD


	(* Internal method *)
	{attribute 'hide'}
	METHOD FB_init : BOOL
	VAR_INPUT
		(*  if TRUE, the retain variables are initialized (warm start / cold start) *)
		bInitRetains : BOOL;
		(*  if TRUE, the instance afterwards gets moved into the copy code (online change) *)
		bInCopyCode : BOOL;
	END_VAR
END_METHOD

END_FUNCTION_BLOCK

// Function Blocks/File Access/FB_VN_WriteContainer

	{attribute 'c++_compatible'}
	{attribute 'external_name' := 'FB_VN_WriteContainer_GUID_398832D9_6000_34F8_0E2A_94AE3FB59320'}
	{attribute 'TcIecLibraryType'}
	(* This FB writes a container as an xml file to the hard drive. *)
	FUNCTION_BLOCK FB_VN_WriteContainer
	VAR_INPUT
		(* The container to write *)
		 {attribute 'GUID' := 'BC72B333-E095-465B-9693-7979773CA3B8'}
		ipContainer : REFERENCE TO ITcVnContainer;
	END_VAR
	VAR_IN_OUT CONSTANT
		(* Full path of the file or relative path to the default directory on the target pc (e.g. only a file name). If the string is empty, a file name will be generated (containing the current time). *)
		 {attribute 'GUID' := '18071995-0000-0000-0000-00000000001A'}
		sFilePath : STRING;
	END_VAR
	VAR_INPUT
		(* Container export format (default is human readable xml) *)
		 {attribute 'GUID' := 'F8305D79-70A3-4F93-A939-2FF3B8D6AF74'}
		 {attribute 'Namespace' := 'Tc3_Vision'}
		eExportFormat : ETcVnContainerExportFormat := TCVN_CEF_XML;
		(* Writing the container is triggered by a rising edge at this input. *)
		bWrite : BOOL;
	END_VAR
	VAR
		 {attribute 'hide'}
		_reserved1 : USINT;
	END_VAR
	VAR_INPUT
		(* Indicates the time before the function is cancelled. *)
		nTimeout : TIME := VISION_ADS_TIMEOUT;
	END_VAR
	VAR_OUTPUT
		(* This output remains TRUE until the function block has executed a command, but at the longest for the duration supplied to the 'nTimeout' input. While bBusy = TRUE, no new command will be accepted at the inputs. *)
		bBusy : BOOL;
		(* This output is switched to TRUE as soon as an error occurs during the execution of a command. The command-specific error code is contained in ‘nErrorId’. If the function block has a timeout error, 'bError' is TRUE and 'nErrorId' is 1861 (hexadecimal 0x745). Is reset to FALSE by the execution of a command at the inputs. *)
		bError : BOOL;
	END_VAR
	VAR
		 {attribute 'hide'}
		_reserved2 : UINT;
	END_VAR
	VAR_OUTPUT
		(* Contains the ADS error code or the command-specific error code of the last executed command. Is reset to 0 by the execution of a command at the inputs. *)
		nErrorId : UDINT;
	END_VAR
	VAR
		(* Internal parameter *)
		{attribute 'hide'}
		nAdsInvStamp : UINT;
		(* Internal parameter *)
		{attribute 'hide'}
		nAdsInvCnt : BYTE;
		 {attribute 'hide'}
		_reserved3 : USINT;
		(* Internal parameter *)
		{attribute 'hide'}
		nTimeElapsed : TIME;
		(* Internal parameter *)
		{attribute 'hide'}
		bLastWrite : BOOL;
		 {attribute 'hide'}
		_reserved4 : UINT_24_56;
	END_VAR


	(* Internal method *)
	{attribute 'hide'}
	METHOD FB_exit : BOOL
	VAR_INPUT
		(* If TRUE, the exit method is called for exiting an instance that is copied afterwards (online change). *)
		bInCopyCode : BOOL;
	END_VAR
END_METHOD


	(* Internal method *)
	{attribute 'hide'}
	METHOD FB_init : BOOL
	VAR_INPUT
		(* If TRUE, the retain variables are initialized (warm start / cold start) *)
		bInitRetains : BOOL;
		(* If TRUE, the instance afterwards gets moved into the copy code (online change) *)
		bInCopyCode : BOOL;
	END_VAR
END_METHOD

END_FUNCTION_BLOCK

// Function Blocks/File Access/FB_VN_WriteImage

	{attribute 'c++_compatible'}
	{attribute 'external_name' := 'FB_VN_WriteImage_GUID_D78879F7_FB0B_383F_0FF9_207E1DA02875'}
	{attribute 'TcIecLibraryType'}
	(* This FB writes an image to the hard drive. *)
	FUNCTION_BLOCK FB_VN_WriteImage
	VAR_INPUT
		(* The image to write *)
		 {attribute 'GUID' := '70D42C6D-6F4E-4719-8B29-2883D5D59B1C'}
		ipImage : REFERENCE TO ITcVnImage;
	END_VAR
	VAR_IN_OUT CONSTANT
		(* Full path of the file or relative path to the default directory on the target pc (e.g. only a file name). If the string is empty, a file name will be generated (containing the current time). *)
		 {attribute 'GUID' := '18071995-0000-0000-0000-00000000001A'}
		sFilePath : STRING;
	END_VAR
	VAR_INPUT
		(* Writing the image is triggered by a rising edge at this input. *)
		bWrite : BOOL;
	END_VAR
	VAR
		 {attribute 'hide'}
		_reserved1 : ARRAY [1..3] OF USINT;
	END_VAR
	VAR_INPUT
		(* Indicates the time before the function is cancelled. *)
		nTimeout : TIME := VISION_ADS_TIMEOUT;
	END_VAR
	VAR_OUTPUT
		(* This output remains TRUE until the function block has executed a command, but at the longest for the duration supplied to the 'nTimeout' input. While bBusy = TRUE, no new command will be accepted at the inputs. *)
		bBusy : BOOL;
		(* This output is switched to TRUE as soon as an error occurs during the execution of a command. The command-specific error code is contained in ‘nErrorId’. If the function block has a timeout error, 'bError' is TRUE and 'nErrorId' is 1861 (hexadecimal 0x745). Is reset to FALSE by the execution of a command at the inputs. *)
		bError : BOOL;
	END_VAR
	VAR
		 {attribute 'hide'}
		_reserved2 : UINT;
	END_VAR
	VAR_OUTPUT
		(* Contains the ADS error code or the command-specific error code of the last executed command. Is reset to 0 by the execution of a command at the inputs. *)
		nErrorId : UDINT;
	END_VAR
	VAR
		(* Internal parameter *)
		{attribute 'hide'}
		nAdsInvStamp : UINT;
		(* Internal parameter *)
		{attribute 'hide'}
		nAdsInvCnt : BYTE;
		 {attribute 'hide'}
		_reserved3 : USINT;
		(* Internal parameter *)
		{attribute 'hide'}
		nTimeElapsed : TIME;
		(* Internal parameter *)
		{attribute 'hide'}
		bLastWrite : BOOL;
		 {attribute 'hide'}
		_reserved4 : UINT_24_56;
	END_VAR


	(* Internal method *)
	{attribute 'hide'}
	METHOD FB_exit : BOOL
	VAR_INPUT
		(*  if TRUE, the exit method is called for exiting an instance that is copied afterwards (online change). *)
		bInCopyCode : BOOL;
	END_VAR
END_METHOD


	(* Internal method *)
	{attribute 'hide'}
	METHOD FB_init : BOOL
	VAR_INPUT
		(*  if TRUE, the retain variables are initialized (warm start / cold start) *)
		bInitRetains : BOOL;
		(*  if TRUE, the instance afterwards gets moved into the copy code (online change) *)
		bInCopyCode : BOOL;
	END_VAR
END_METHOD

END_FUNCTION_BLOCK

// Function Blocks/File Access/FB_VN_WriteMlModel

	{attribute 'c++_compatible'}
	{attribute 'external_name' := 'FB_VN_WriteMlModel_GUID_59C743C5_5507_31C7_2AE8_C3C8D0109762'}
	{attribute 'TcIecLibraryType'}
	(* This FB writes a machine learning model to the hard drive. *)
	FUNCTION_BLOCK FB_VN_WriteMlModel
	VAR_INPUT
		(* The machine learning model to write *)
		 {attribute 'GUID' := 'AC23D64B-CDFA-4D43-AE8B-364A856EB3E2'}
		ipMlModel : REFERENCE TO ITcVnMlModel;
	END_VAR
	VAR_IN_OUT CONSTANT
		(* Full path of the file or relative path to the default directory on the target pc (e.g. only a file name). If the string is empty, a file name will be generated (containing the current time). *)
		 {attribute 'GUID' := '18071995-0000-0000-0000-00000000001A'}
		sFilePath : STRING;
	END_VAR
	VAR_INPUT
		(* Writing the machine learning model is triggered by a rising edge at this input. *)
		bWrite : BOOL;
	END_VAR
	VAR
		 {attribute 'hide'}
		_reserved1 : ARRAY [1..3] OF USINT;
	END_VAR
	VAR_INPUT
		(* Indicates the time before the function is cancelled. *)
		nTimeout : TIME := VISION_ADS_TIMEOUT;
	END_VAR
	VAR_OUTPUT
		(* This output remains TRUE until the function block has executed a command, but at the longest for the duration supplied to the 'nTimeout' input. While bBusy = TRUE, no new command will be accepted at the inputs. *)
		bBusy : BOOL;
		(* This output is switched to TRUE as soon as an error occurs during the execution of a command. The command-specific error code is contained in ‘nErrorId’. If the function block has a timeout error, 'bError' is TRUE and 'nErrorId' is 1861 (hexadecimal 0x745). Is reset to FALSE by the execution of a command at the inputs. *)
		bError : BOOL;
	END_VAR
	VAR
		 {attribute 'hide'}
		_reserved2 : UINT;
	END_VAR
	VAR_OUTPUT
		(* Contains the ADS error code or the command-specific error code of the last executed command. Is reset to 0 by the execution of a command at the inputs. *)
		nErrorId : UDINT;
	END_VAR
	VAR
		(* Internal parameter *)
		{attribute 'hide'}
		nAdsInvStamp : UINT;
		(* Internal parameter *)
		{attribute 'hide'}
		nAdsInvCnt : BYTE;
		 {attribute 'hide'}
		_reserved3 : USINT;
		(* Internal parameter *)
		{attribute 'hide'}
		nTimeElapsed : TIME;
		(* Internal parameter *)
		{attribute 'hide'}
		bLastWrite : BOOL;
		 {attribute 'hide'}
		_reserved4 : UINT_24_56;
	END_VAR


	(* Internal method *)
	{attribute 'hide'}
	METHOD FB_exit : BOOL
	VAR_INPUT
		(*  if TRUE, the exit method is called for exiting an instance that is copied afterwards (online change). *)
		bInCopyCode : BOOL;
	END_VAR
END_METHOD


	(* Internal method *)
	{attribute 'hide'}
	METHOD FB_init : BOOL
	VAR_INPUT
		(*  if TRUE, the retain variables are initialized (warm start / cold start) *)
		bInitRetains : BOOL;
		(*  if TRUE, the instance afterwards gets moved into the copy code (online change) *)
		bInCopyCode : BOOL;
	END_VAR
END_METHOD

END_FUNCTION_BLOCK

// Function Blocks/Camera Register Access/FB_VN_ReadRegister_UDINT

	{attribute 'c++_compatible'}
	{attribute 'external_name' := 'FB_VN_ReadRegister_UDINT_GUID_C67D4C63_2EDC_3714_1279_ABD9F7DF7AD0'}
	{attribute 'TcIecLibraryType'}
	(* This FB reads a DINT register from the camera. Requires an open control channel (e.g. by calling FB_VN_GevCameraControl.OpenCamera() before) *)
	FUNCTION_BLOCK FB_VN_ReadRegister_UDINT
	VAR_INPUT
		(* The address of the register that should be read *)
		 {attribute 'GUID' := 'E1ED2436-3512-43FA-B927-3F71DEDDA853'}
		nAddress : GVCP_REGISTER_ADDRESS;
		(* OPTIONAL: The endianness of the register. 0 = Big, 1 = Little. Default: 0 *)
		nEndian : UINT;
		(* Reading the register is triggered by a rising edge at this input. *)
		bRead : BOOL;
	END_VAR
	VAR
		 {attribute 'hide'}
		_reserved1 : USINT;
	END_VAR
	VAR_INPUT
		(* Indicates the time before the function is cancelled. *)
		nTimeout : TIME := VISION_ADS_TIMEOUT;
	END_VAR
	VAR_OUTPUT
		(* The read value *)
		nValue : UDINT;
		(* This output remains TRUE until the function block has executed a command, but at the longest for the duration supplied to the 'nTimeout' input. While bBusy = TRUE, no new command will be accepted at the inputs. *)
		bBusy : BOOL;
		(* This output is switched to TRUE as soon as an error occurs during the execution of a command. The command-specific error code is contained in ‘nErrorId’. If the function block has a timeout error, 'bError' is TRUE and 'nErrorId' is 1861 (hexadecimal 0x745). Is reset to FALSE by the execution of a command at the inputs. *)
		bError : BOOL;
	END_VAR
	VAR
		 {attribute 'hide'}
		_reserved2 : UINT;
	END_VAR
	VAR_OUTPUT
		(* Contains the ADS error code or the command-specific error code of the last executed command. Is reset to 0 by the execution of a command at the inputs. *)
		nErrorId : UDINT;
	END_VAR
	VAR
		(* Internal reference to the corresponding TcVnGevImageProvider TcCOM module ID, which needs to be set via TC init symbol. *)
		{attribute 'TcInitSymbol'}
		{attribute 'TcCategoryOID' := 'TcVnGevImageProvider'}
		 {attribute 'GUID' := '18071995-0000-0000-0000-00000000000F'}
		oidITcVnGevImageProvider : OTCID;
		 {attribute 'hide'}
		_reserved3 : UINT_0_32;
		(* Internal reference to the corresponding TcVnGevImageProvider module. *)
		{attribute 'hide'}
		 {attribute 'GUID' := 'ED7659DB-95DC-4A4A-B62F-02C9870D5E81'}
		ipGevImageProvider : ITcVnGevImageProvider;
		(* Internal timestamp for timeout detection *)
		{attribute 'hide'}
		nTimeElapsed : TIME;
		(* Internal flag for rising edge detection *)
		{attribute 'hide'}
		bLastRead : BOOL;
		 {attribute 'hide'}
		_reserved4 : ARRAY [1..3] OF USINT;
	END_VAR


	(* Internal method *)
	{attribute 'hide'}
	METHOD FB_exit : BOOL
	VAR_INPUT
		(*  if TRUE, the exit method is called for exiting an instance that is copied afterwards (online change). *)
		bInCopyCode : BOOL;
	END_VAR
END_METHOD


	(* Internal method *)
	{attribute 'hide'}
	METHOD FB_init : BOOL
	VAR_INPUT
		(*  if TRUE, the retain variables are initialized (warm start / cold start) *)
		bInitRetains : BOOL;
		(*  if TRUE, the instance afterwards gets moved into the copy code (online change) *)
		bInCopyCode : BOOL;
	END_VAR
END_METHOD

END_FUNCTION_BLOCK

// Function Blocks/Camera Register Access/FB_VN_WriteRegister_UDINT

	{attribute 'c++_compatible'}
	{attribute 'external_name' := 'FB_VN_WriteRegister_UDINT_GUID_D8217EFB_F59F_3DB6_0CBB_C513551B9472'}
	{attribute 'TcIecLibraryType'}
	(* This FB writes a DINT value into a register on the camera. Requires an open control channel (e.g. by calling FB_VN_GevCameraControl.OpenCamera() before) *)
	FUNCTION_BLOCK FB_VN_WriteRegister_UDINT
	VAR_INPUT
		(* The address of the register that should be written *)
		 {attribute 'GUID' := 'E1ED2436-3512-43FA-B927-3F71DEDDA853'}
		nAddress : GVCP_REGISTER_ADDRESS;
		(* The value to write *)
		nValue : UDINT;
		(* OPTIONAL: The endianness of the register. 0 = Big, 1 = Little. Default: 0 *)
		nEndian : UINT;
		(* Reading the register is triggered by a rising edge at this input. *)
		bWrite : BOOL;
	END_VAR
	VAR
		 {attribute 'hide'}
		_reserved1 : USINT;
	END_VAR
	VAR_INPUT
		(* Indicates the time before the function is cancelled. *)
		nTimeout : TIME := VISION_ADS_TIMEOUT;
	END_VAR
	VAR_OUTPUT
		(* This output remains TRUE until the function block has executed a command, but at the longest for the duration supplied to the 'nTimeout' input. While bBusy = TRUE, no new command will be accepted at the inputs. *)
		bBusy : BOOL;
		(* This output is switched to TRUE as soon as an error occurs during the execution of a command. The command-specific error code is contained in ‘nErrorId’. If the function block has a timeout error, 'bError' is TRUE and 'nErrorId' is 1861 (hexadecimal 0x745). Is reset to FALSE by the execution of a command at the inputs. *)
		bError : BOOL;
	END_VAR
	VAR
		 {attribute 'hide'}
		_reserved2 : UINT;
	END_VAR
	VAR_OUTPUT
		(* Contains the ADS error code or the command-specific error code of the last executed command. Is reset to 0 by the execution of a command at the inputs. *)
		nErrorId : UDINT;
	END_VAR
	VAR
		(* Internal reference to the corresponding TcVnGevImageProvider TcCOM module ID, which needs to be set via TC init symbol. *)
		{attribute 'TcInitSymbol'}
		{attribute 'TcCategoryOID' := 'TcVnGevImageProvider'}
		 {attribute 'GUID' := '18071995-0000-0000-0000-00000000000F'}
		oidITcVnGevImageProvider : OTCID;
		 {attribute 'hide'}
		_reserved3 : UINT_0_32;
		(* Internal reference to the corresponding TcVnGevImageProvider module. *)
		{attribute 'hide'}
		 {attribute 'GUID' := 'ED7659DB-95DC-4A4A-B62F-02C9870D5E81'}
		ipGevImageProvider : ITcVnGevImageProvider;
		(* Internal timestamp for timeout detection *)
		{attribute 'hide'}
		nTimeElapsed : TIME;
		(* Internal flag for rising edge detection *)
		{attribute 'hide'}
		bLastWrite : BOOL;
		 {attribute 'hide'}
		_reserved4 : ARRAY [1..3] OF USINT;
	END_VAR


	(* Internal method *)
	{attribute 'hide'}
	METHOD FB_exit : BOOL
	VAR_INPUT
		(*  if TRUE, the exit method is called for exiting an instance that is copied afterwards (online change). *)
		bInCopyCode : BOOL;
	END_VAR
END_METHOD


	(* Internal method *)
	{attribute 'hide'}
	METHOD FB_init : BOOL
	VAR_INPUT
		(*  if TRUE, the retain variables are initialized (warm start / cold start) *)
		bInitRetains : BOOL;
		(*  if TRUE, the instance afterwards gets moved into the copy code (online change) *)
		bInCopyCode : BOOL;
	END_VAR
END_METHOD

END_FUNCTION_BLOCK

// Function Blocks/Camera Register Access/FB_VN_ReadRegister_ULINT

	{attribute 'c++_compatible'}
	{attribute 'external_name' := 'FB_VN_ReadRegister_ULINT_GUID_1A2FF669_1438_39FC_19FC_4114B90D0335'}
	{attribute 'TcIecLibraryType'}
	(* This FB reads a ULINT register from the camera. Requires an open control channel (e.g. by calling FB_VN_GevCameraControl.OpenCamera() before) *)
	FUNCTION_BLOCK FB_VN_ReadRegister_ULINT
	VAR_INPUT
		(* The address of the register that should be read *)
		 {attribute 'GUID' := 'E1ED2436-3512-43FA-B927-3F71DEDDA853'}
		nAddress : GVCP_REGISTER_ADDRESS;
		(* OPTIONAL: The endianness of the register. 0 = Big, 1 = Little. Default: 0 *)
		nEndian : UINT;
		(* Reading the register is triggered by a rising edge at this input. *)
		bRead : BOOL;
	END_VAR
	VAR
		 {attribute 'hide'}
		_reserved1 : USINT;
	END_VAR
	VAR_INPUT
		(* Indicates the time before the function is cancelled. *)
		nTimeout : TIME := VISION_ADS_TIMEOUT;
	END_VAR
	VAR
		 {attribute 'hide'}
		_reserved2 : UINT_0_32;
	END_VAR
	VAR_OUTPUT
		(* The read value *)
		nValue : ULINT;
		(* This output remains TRUE until the function block has executed a command, but at the longest for the duration supplied to the 'nTimeout' input. While bBusy = TRUE, no new command will be accepted at the inputs. *)
		bBusy : BOOL;
		(* This output is switched to TRUE as soon as an error occurs during the execution of a command. The command-specific error code is contained in ‘nErrorId’. If the function block has a timeout error, 'bError' is TRUE and 'nErrorId' is 1861 (hexadecimal 0x745). Is reset to FALSE by the execution of a command at the inputs. *)
		bError : BOOL;
	END_VAR
	VAR
		 {attribute 'hide'}
		_reserved3 : UINT;
	END_VAR
	VAR_OUTPUT
		(* Contains the ADS error code or the command-specific error code of the last executed command. Is reset to 0 by the execution of a command at the inputs. *)
		nErrorId : UDINT;
	END_VAR
	VAR
		(* Internal reference to the corresponding TcVnGevImageProvider TcCOM module ID, which needs to be set via TC init symbol. *)
		{attribute 'TcInitSymbol'}
		{attribute 'TcCategoryOID' := 'TcVnGevImageProvider'}
		 {attribute 'GUID' := '18071995-0000-0000-0000-00000000000F'}
		oidITcVnGevImageProvider : OTCID;
		 {attribute 'hide'}
		_reserved4 : UINT_0_32;
		(* Internal reference to the corresponding TcVnGevImageProvider module. *)
		{attribute 'hide'}
		 {attribute 'GUID' := 'ED7659DB-95DC-4A4A-B62F-02C9870D5E81'}
		ipGevImageProvider : ITcVnGevImageProvider;
		(* Internal timestamp for timeout detection *)
		{attribute 'hide'}
		nTimeElapsed : TIME;
		(* Internal flag for rising edge detection *)
		{attribute 'hide'}
		bLastRead : BOOL;
		 {attribute 'hide'}
		_reserved5 : ARRAY [1..3] OF USINT;
	END_VAR


	(* Internal method *)
	{attribute 'hide'}
	METHOD FB_exit : BOOL
	VAR_INPUT
		(*  if TRUE, the exit method is called for exiting an instance that is copied afterwards (online change). *)
		bInCopyCode : BOOL;
	END_VAR
END_METHOD


	(* Internal method *)
	{attribute 'hide'}
	METHOD FB_init : BOOL
	VAR_INPUT
		(*  if TRUE, the retain variables are initialized (warm start / cold start) *)
		bInitRetains : BOOL;
		(*  if TRUE, the instance afterwards gets moved into the copy code (online change) *)
		bInCopyCode : BOOL;
	END_VAR
END_METHOD

END_FUNCTION_BLOCK

// Function Blocks/Camera Register Access/FB_VN_WriteRegister_ULINT

	{attribute 'c++_compatible'}
	{attribute 'external_name' := 'FB_VN_WriteRegister_ULINT_GUID_8279FD7F_D5C2_35EF_30D0_3125E29E2C03'}
	{attribute 'TcIecLibraryType'}
	(* This FB writes a ULINT value into a register on the camera. Requires an open control channel (e.g. by calling FB_VN_GevCameraControl.OpenCamera() before) *)
	FUNCTION_BLOCK FB_VN_WriteRegister_ULINT
	VAR_INPUT
		(* The address of the register that should be written *)
		 {attribute 'GUID' := 'E1ED2436-3512-43FA-B927-3F71DEDDA853'}
		nAddress : GVCP_REGISTER_ADDRESS;
	END_VAR
	VAR
		 {attribute 'hide'}
		_reserved1 : UINT_0_32;
	END_VAR
	VAR_INPUT
		(* The value to write *)
		nValue : ULINT;
		(* OPTIONAL: The endianness of the register. 0 = Big, 1 = Little. Default: 0 *)
		nEndian : UINT;
		(* Reading the register is triggered by a rising edge at this input. *)
		bWrite : BOOL;
	END_VAR
	VAR
		 {attribute 'hide'}
		_reserved2 : USINT;
	END_VAR
	VAR_INPUT
		(* Indicates the time before the function is cancelled. *)
		nTimeout : TIME := VISION_ADS_TIMEOUT;
	END_VAR
	VAR_OUTPUT
		(* This output remains TRUE until the function block has executed a command, but at the longest for the duration supplied to the 'nTimeout' input. While bBusy = TRUE, no new command will be accepted at the inputs. *)
		bBusy : BOOL;
		(* This output is switched to TRUE as soon as an error occurs during the execution of a command. The command-specific error code is contained in ‘nErrorId’. If the function block has a timeout error, 'bError' is TRUE and 'nErrorId' is 1861 (hexadecimal 0x745). Is reset to FALSE by the execution of a command at the inputs. *)
		bError : BOOL;
	END_VAR
	VAR
		 {attribute 'hide'}
		_reserved3 : UINT;
	END_VAR
	VAR_OUTPUT
		(* Contains the ADS error code or the command-specific error code of the last executed command. Is reset to 0 by the execution of a command at the inputs. *)
		nErrorId : UDINT;
	END_VAR
	VAR
		(* Internal reference to the corresponding TcVnGevImageProvider TcCOM module ID, which needs to be set via TC init symbol. *)
		{attribute 'TcInitSymbol'}
		{attribute 'TcCategoryOID' := 'TcVnGevImageProvider'}
		 {attribute 'GUID' := '18071995-0000-0000-0000-00000000000F'}
		oidITcVnGevImageProvider : OTCID;
		 {attribute 'hide'}
		_reserved4 : UINT_0_32;
		(* Internal reference to the corresponding TcVnGevImageProvider module. *)
		{attribute 'hide'}
		 {attribute 'GUID' := 'ED7659DB-95DC-4A4A-B62F-02C9870D5E81'}
		ipGevImageProvider : ITcVnGevImageProvider;
		(* Internal timestamp for timeout detection *)
		{attribute 'hide'}
		nTimeElapsed : TIME;
		(* Internal flag for rising edge detection *)
		{attribute 'hide'}
		bLastWrite : BOOL;
		 {attribute 'hide'}
		_reserved5 : ARRAY [1..3] OF USINT;
	END_VAR


	(* Internal method *)
	{attribute 'hide'}
	METHOD FB_exit : BOOL
	VAR_INPUT
		(*  if TRUE, the exit method is called for exiting an instance that is copied afterwards (online change). *)
		bInCopyCode : BOOL;
	END_VAR
END_METHOD


	(* Internal method *)
	{attribute 'hide'}
	METHOD FB_init : BOOL
	VAR_INPUT
		(*  if TRUE, the retain variables are initialized (warm start / cold start) *)
		bInitRetains : BOOL;
		(*  if TRUE, the instance afterwards gets moved into the copy code (online change) *)
		bInCopyCode : BOOL;
	END_VAR
END_METHOD

END_FUNCTION_BLOCK

// Function Blocks/Camera Register Access/FB_VN_ReadMemory

	{attribute 'c++_compatible'}
	{attribute 'external_name' := 'FB_VN_ReadMemory_GUID_EB04D561_C27C_3BB7_2B6A_FDA13CCE2D83'}
	{attribute 'TcIecLibraryType'}
	(* This FB reads consecutive memory locations from the camera. Requires an open control channel (e.g. by calling FB_VN_GevCameraControl.OpenCamera() before) *)
	FUNCTION_BLOCK FB_VN_ReadMemory
	VAR_INPUT
		(* The address of the first byte to read from the camera (must be 32-bit aligned) *)
		 {attribute 'GUID' := 'E1ED2436-3512-43FA-B927-3F71DEDDA853'}
		nAddress : GVCP_REGISTER_ADDRESS;
		(* The number of bytes to read, starting with nAddress (must be a multiple of 4, not more than 536) *)
		nLength : UINT;
	END_VAR
	VAR
		 {attribute 'hide'}
		_reserved1 : UINT;
	END_VAR
	VAR_INPUT
		(* Pointer to the buffer where the read memory content is written to (The buffer must have a size of at least nLength bytes!) *)
		 {attribute 'GUID' := '18071995-0000-0000-0000-000000000018'}
		pBuffer : PVOID;
		(* Reading the memory is triggered by a rising edge at this input. *)
		bRead : BOOL;
	END_VAR
	VAR
		 {attribute 'hide'}
		_reserved2 : ARRAY [1..3] OF USINT;
	END_VAR
	VAR_INPUT
		(* Indicates the time before the function is cancelled. *)
		nTimeout : TIME := VISION_ADS_TIMEOUT;
	END_VAR
	VAR_OUTPUT
		(* This output remains TRUE until the function block has executed a command, but at the longest for the duration supplied to the 'nTimeout' input. While bBusy = TRUE, no new command will be accepted at the inputs. *)
		bBusy : BOOL;
		(* This output is switched to TRUE as soon as an error occurs during the execution of a command. The command-specific error code is contained in ‘nErrorId’. If the function block has a timeout error, 'bError' is TRUE and 'nErrorId' is 1861 (hexadecimal 0x745). Is reset to FALSE by the execution of a command at the inputs. *)
		bError : BOOL;
	END_VAR
	VAR
		 {attribute 'hide'}
		_reserved3 : UINT;
	END_VAR
	VAR_OUTPUT
		(* Contains the ADS error code or the command-specific error code of the last executed command. Is reset to 0 by the execution of a command at the inputs. *)
		nErrorId : UDINT;
	END_VAR
	VAR
		(* Internal reference to the corresponding TcVnGevImageProvider TcCOM module ID, which needs to be set via TC init symbol. *)
		{attribute 'TcInitSymbol'}
		{attribute 'TcCategoryOID' := 'TcVnGevImageProvider'}
		 {attribute 'GUID' := '18071995-0000-0000-0000-00000000000F'}
		oidITcVnGevImageProvider : OTCID;
		 {attribute 'hide'}
		_reserved4 : UINT_0_32;
		(* Internal reference to the corresponding TcVnGevImageProvider module. *)
		{attribute 'hide'}
		 {attribute 'GUID' := 'ED7659DB-95DC-4A4A-B62F-02C9870D5E81'}
		ipGevImageProvider : ITcVnGevImageProvider;
		(* Internal timestamp for timeout detection *)
		{attribute 'hide'}
		nTimeElapsed : TIME;
		(* Internal flag for rising edge detection *)
		{attribute 'hide'}
		bLastRead : BOOL;
		 {attribute 'hide'}
		_reserved5 : ARRAY [1..3] OF USINT;
	END_VAR


	(* Internal method *)
	{attribute 'hide'}
	METHOD FB_exit : BOOL
	VAR_INPUT
		(* If TRUE, the exit method is called for exiting an instance that is copied afterwards (online change). *)
		bInCopyCode : BOOL;
	END_VAR
END_METHOD


	(* Internal method *)
	{attribute 'hide'}
	METHOD FB_init : BOOL
	VAR_INPUT
		(* If TRUE, the retain variables are initialized (warm start / cold start) *)
		bInitRetains : BOOL;
		(* If TRUE, the instance afterwards gets moved into the copy code (online change) *)
		bInCopyCode : BOOL;
	END_VAR
END_METHOD

END_FUNCTION_BLOCK

// Function Blocks/Camera Register Access/FB_VN_WriteMemory

	{attribute 'c++_compatible'}
	{attribute 'external_name' := 'FB_VN_WriteMemory_GUID_FE24C77B_8B65_3093_38E1_349A728AAFD6'}
	{attribute 'TcIecLibraryType'}
	(* This FB writes data to consecutive memory locations on the camera. Requires an open control channel (e.g. by calling FB_VN_GevCameraControl.OpenCamera() before) *)
	FUNCTION_BLOCK FB_VN_WriteMemory
	VAR_INPUT
		(* The address of the first byte to write to the camera (must be 32-bit aligned) *)
		 {attribute 'GUID' := 'E1ED2436-3512-43FA-B927-3F71DEDDA853'}
		nAddress : GVCP_REGISTER_ADDRESS;
		(* The number of bytes to write, starting at nAddress (must be a multiple of 4, not more than 536) *)
		nLength : UINT;
	END_VAR
	VAR
		 {attribute 'hide'}
		_reserved1 : UINT;
	END_VAR
	VAR_INPUT
		(* Pointer to the data that should be written to the camera (must have a size of at least nLength bytes!) *)
		 {attribute 'GUID' := '18071995-0000-0000-0000-000000000018'}
		pData : PVOID;
		(* Writing the memory is triggered by a rising edge at this input. *)
		bWrite : BOOL;
	END_VAR
	VAR
		 {attribute 'hide'}
		_reserved2 : ARRAY [1..3] OF USINT;
	END_VAR
	VAR_INPUT
		(* Indicates the time before the function is cancelled. *)
		nTimeout : TIME := VISION_ADS_TIMEOUT;
	END_VAR
	VAR_OUTPUT
		(* This output remains TRUE until the function block has executed a command, but at the longest for the duration supplied to the 'nTimeout' input. While bBusy = TRUE, no new command will be accepted at the inputs. *)
		bBusy : BOOL;
		(* This output is switched to TRUE as soon as an error occurs during the execution of a command. The command-specific error code is contained in ‘nErrorId’. If the function block has a timeout error, 'bError' is TRUE and 'nErrorId' is 1861 (hexadecimal 0x745). Is reset to FALSE by the execution of a command at the inputs. *)
		bError : BOOL;
	END_VAR
	VAR
		 {attribute 'hide'}
		_reserved3 : UINT;
	END_VAR
	VAR_OUTPUT
		(* Contains the ADS error code or the command-specific error code of the last executed command. Is reset to 0 by the execution of a command at the inputs. *)
		nErrorId : UDINT;
		(* The number of bytes that have been successfully written to the camera. *)
		nBytesWritten : UINT;
	END_VAR
	VAR
		 {attribute 'hide'}
		_reserved4 : UINT;
		(* Internal reference to the corresponding TcVnGevImageProvider TcCOM module ID, which needs to be set via TC init symbol. *)
		{attribute 'TcInitSymbol'}
		{attribute 'TcCategoryOID' := 'TcVnGevImageProvider'}
		 {attribute 'GUID' := '18071995-0000-0000-0000-00000000000F'}
		oidITcVnGevImageProvider : OTCID;
		(* Internal reference to the corresponding TcVnGevImageProvider module. *)
		{attribute 'hide'}
		 {attribute 'GUID' := 'ED7659DB-95DC-4A4A-B62F-02C9870D5E81'}
		ipGevImageProvider : ITcVnGevImageProvider;
		(* Internal timestamp for timeout detection *)
		{attribute 'hide'}
		nTimeElapsed : TIME;
		(* Internal flag for rising edge detection *)
		{attribute 'hide'}
		bLastRead : BOOL;
		 {attribute 'hide'}
		_reserved5 : ARRAY [1..3] OF USINT;
	END_VAR


	(* Internal method *)
	{attribute 'hide'}
	METHOD FB_exit : BOOL
	VAR_INPUT
		(* If TRUE, the exit method is called for exiting an instance that is copied afterwards (online change). *)
		bInCopyCode : BOOL;
	END_VAR
END_METHOD


	(* Internal method *)
	{attribute 'hide'}
	METHOD FB_init : BOOL
	VAR_INPUT
		(* If TRUE, the retain variables are initialized (warm start / cold start) *)
		bInitRetains : BOOL;
		(* If TRUE, the instance afterwards gets moved into the copy code (online change) *)
		bInCopyCode : BOOL;
	END_VAR
END_METHOD

END_FUNCTION_BLOCK

// Function Blocks/Camera Register Access/FB_VN_ReadRegister_REAL

	{attribute 'c++_compatible'}
	{attribute 'external_name' := 'FB_VN_ReadRegister_REAL_GUID_9C3EF46F_45EB_34DB_2434_F59855585573'}
	{attribute 'TcIecLibraryType'}
	(* This FB reads a REAL register from the camera. Requires an open control channel (e.g. by calling FB_VN_GevCameraControl.OpenCamera() before) *)
	FUNCTION_BLOCK FB_VN_ReadRegister_REAL
	VAR_INPUT
		(* The address of the register that should be read *)
		 {attribute 'GUID' := 'E1ED2436-3512-43FA-B927-3F71DEDDA853'}
		nAddress : GVCP_REGISTER_ADDRESS;
		(* OPTIONAL: The endianness of the register. 0 = Big, 1 = Little. Default: 0 *)
		nEndian : UINT;
		(* Reading the register is triggered by a rising edge at this input. *)
		bRead : BOOL;
	END_VAR
	VAR
		 {attribute 'hide'}
		_reserved1 : USINT;
	END_VAR
	VAR_INPUT
		(* Indicates the time before the function is cancelled. *)
		nTimeout : TIME := VISION_ADS_TIMEOUT;
	END_VAR
	VAR_OUTPUT
		(* The read value *)
		fValue : REAL;
		(* This output remains TRUE until the function block has executed a command, but at the longest for the duration supplied to the 'nTimeout' input. While bBusy = TRUE, no new command will be accepted at the inputs. *)
		bBusy : BOOL;
		(* This output is switched to TRUE as soon as an error occurs during the execution of a command. The command-specific error code is contained in ‘nErrorId’. If the function block has a timeout error, 'bError' is TRUE and 'nErrorId' is 1861 (hexadecimal 0x745). Is reset to FALSE by the execution of a command at the inputs. *)
		bError : BOOL;
	END_VAR
	VAR
		 {attribute 'hide'}
		_reserved2 : UINT;
	END_VAR
	VAR_OUTPUT
		(* Contains the ADS error code or the command-specific error code of the last executed command. Is reset to 0 by the execution of a command at the inputs. *)
		nErrorId : UDINT;
	END_VAR
	VAR
		(* Internal reference to the corresponding TcVnGevImageProvider TcCOM module ID, which needs to be set via TC init symbol. *)
		{attribute 'TcInitSymbol'}
		{attribute 'TcCategoryOID' := 'TcVnGevImageProvider'}
		 {attribute 'GUID' := '18071995-0000-0000-0000-00000000000F'}
		oidITcVnGevImageProvider : OTCID;
		 {attribute 'hide'}
		_reserved3 : UINT_0_32;
		(* Internal reference to the corresponding TcVnGevImageProvider module. *)
		{attribute 'hide'}
		 {attribute 'GUID' := 'ED7659DB-95DC-4A4A-B62F-02C9870D5E81'}
		ipGevImageProvider : ITcVnGevImageProvider;
		(* Internal timestamp for timeout detection *)
		{attribute 'hide'}
		nTimeElapsed : TIME;
		(* Internal flag for rising edge detection *)
		{attribute 'hide'}
		bLastRead : BOOL;
		 {attribute 'hide'}
		_reserved4 : ARRAY [1..3] OF USINT;
	END_VAR


	(* Internal method *)
	{attribute 'hide'}
	METHOD FB_exit : BOOL
	VAR_INPUT
		(*  if TRUE, the exit method is called for exiting an instance that is copied afterwards (online change). *)
		bInCopyCode : BOOL;
	END_VAR
END_METHOD


	(* Internal method *)
	{attribute 'hide'}
	METHOD FB_init : BOOL
	VAR_INPUT
		(*  if TRUE, the retain variables are initialized (warm start / cold start) *)
		bInitRetains : BOOL;
		(*  if TRUE, the instance afterwards gets moved into the copy code (online change) *)
		bInCopyCode : BOOL;
	END_VAR
END_METHOD

END_FUNCTION_BLOCK

// Function Blocks/Camera Register Access/FB_VN_WriteRegister_REAL

	{attribute 'c++_compatible'}
	{attribute 'external_name' := 'FB_VN_WriteRegister_REAL_GUID_8B382016_C297_3DA8_21DF_E9A51DAFA566'}
	{attribute 'TcIecLibraryType'}
	(* This FB writes a REAL value into a register on the camera. Requires an open control channel (e.g. by calling FB_VN_GevCameraControl.OpenCamera() before) *)
	FUNCTION_BLOCK FB_VN_WriteRegister_REAL
	VAR_INPUT
		(* The address of the register that should be written *)
		 {attribute 'GUID' := 'E1ED2436-3512-43FA-B927-3F71DEDDA853'}
		nAddress : GVCP_REGISTER_ADDRESS;
		(* The value to write *)
		fValue : REAL;
		(* OPTIONAL: The endianness of the register. 0 = Big, 1 = Little. Default: 0 *)
		nEndian : UINT;
		(* Writing the register is triggered by a rising edge at this input. *)
		bWrite : BOOL;
	END_VAR
	VAR
		 {attribute 'hide'}
		_reserved1 : USINT;
	END_VAR
	VAR_INPUT
		(* Indicates the time before the function is cancelled. *)
		nTimeout : TIME := VISION_ADS_TIMEOUT;
	END_VAR
	VAR_OUTPUT
		(* This output remains TRUE until the function block has executed a command, but at the longest for the duration supplied to the 'nTimeout' input. While bBusy = TRUE, no new command will be accepted at the inputs. *)
		bBusy : BOOL;
		(* This output is switched to TRUE as soon as an error occurs during the execution of a command. The command-specific error code is contained in ‘nErrorId’. If the function block has a timeout error, 'bError' is TRUE and 'nErrorId' is 1861 (hexadecimal 0x745). Is reset to FALSE by the execution of a command at the inputs. *)
		bError : BOOL;
	END_VAR
	VAR
		 {attribute 'hide'}
		_reserved2 : UINT;
	END_VAR
	VAR_OUTPUT
		(* Contains the ADS error code or the command-specific error code of the last executed command. Is reset to 0 by the execution of a command at the inputs. *)
		nErrorId : UDINT;
	END_VAR
	VAR
		(* Internal reference to the corresponding TcVnGevImageProvider TcCOM module ID, which needs to be set via TC init symbol. *)
		{attribute 'TcInitSymbol'}
		{attribute 'TcCategoryOID' := 'TcVnGevImageProvider'}
		 {attribute 'GUID' := '18071995-0000-0000-0000-00000000000F'}
		oidITcVnGevImageProvider : OTCID;
		 {attribute 'hide'}
		_reserved3 : UINT_0_32;
		(* Internal reference to the corresponding TcVnGevImageProvider module. *)
		{attribute 'hide'}
		 {attribute 'GUID' := 'ED7659DB-95DC-4A4A-B62F-02C9870D5E81'}
		ipGevImageProvider : ITcVnGevImageProvider;
		(* Internal timestamp for timeout detection *)
		{attribute 'hide'}
		nTimeElapsed : TIME;
		(* Internal flag for rising edge detection *)
		{attribute 'hide'}
		bLastWrite : BOOL;
		 {attribute 'hide'}
		_reserved4 : ARRAY [1..3] OF USINT;
	END_VAR


	(* Internal method *)
	{attribute 'hide'}
	METHOD FB_exit : BOOL
	VAR_INPUT
		(*  if TRUE, the exit method is called for exiting an instance that is copied afterwards (online change). *)
		bInCopyCode : BOOL;
	END_VAR
END_METHOD


	(* Internal method *)
	{attribute 'hide'}
	METHOD FB_init : BOOL
	VAR_INPUT
		(*  if TRUE, the retain variables are initialized (warm start / cold start) *)
		bInitRetains : BOOL;
		(*  if TRUE, the instance afterwards gets moved into the copy code (online change) *)
		bInCopyCode : BOOL;
	END_VAR
END_METHOD

END_FUNCTION_BLOCK

// Function Blocks/Image Processing/FB_VN_GeneralizedHoughBallard

	{attribute 'c++_compatible'}
	{attribute 'external_name' := 'FB_VN_GeneralizedHoughBallard_GUID_BF79B715_AD91_35EE_0D29_B7631CED420B'}
	{attribute 'TcIecLibraryType'}
	{attribute 'no_explicit_call' :='do not call this POU directly'}
	(* This FB provides the Generalized Hough Ballard functionality. First, set the parameters via the corresponding methods (optional, defaults are used otherwise). Then, set the template (required). Afterwards, the Detect method can be executed. *)
	FUNCTION_BLOCK FB_VN_GeneralizedHoughBallard
	VAR
		(* Internal stuff *)
		{attribute 'hide'}
		 {attribute 'GUID' := '18071995-0000-0000-0000-000000000018'}
		internal1 : PVOID;
		(* Internal stuff *)
		{attribute 'hide'}
		 {attribute 'GUID' := '18071995-0000-0000-0000-000000000018'}
		internal2 : PVOID;
		(* Internal stuff *)
		{attribute 'hide'}
		internal3 : BOOL;
		 {attribute 'hide'}
		_reserved1 : UINT_24_56;
	END_VAR


	(* Internal method *)
	{attribute 'hide'}
	METHOD FB_exit : BOOL
	VAR_INPUT
		(* if TRUE, the exit method is called for exiting an instance that is copied afterwards (online change). *)
		bInCopyCode : BOOL;
	END_VAR
END_METHOD


	(* Internal method *)
	{attribute 'hide'}
	METHOD FB_init : BOOL
	VAR_INPUT
		(* if TRUE, the retain variables are initialized (warm start / cold start) *)
		bInitRetains : BOOL;
		(* if TRUE, the instance afterwards gets moved into the copy code (online change) *)
		bInCopyCode : BOOL;
	END_VAR
END_METHOD


	(* Detect the template in an image (SetTemplate must have been called before). *)
	METHOD Detect : HRESULT
	VAR_INPUT
		(* Source image (1 channel, USINT) *)
 {attribute 'GUID' := '70D42C6D-6F4E-4719-8B29-2883D5D59B1C'}
				ipImage : ITcVnImage;
		(* Returns the centers of the detected template positions (ContainerType_Vector_TcVnPoint2_REAL; Non-zero interface pointers are reused.) *)
 {attribute 'GUID' := 'BC72B333-E095-465B-9693-7979773CA3B8'}
				ipPositions : REFERENCE TO ITcVnContainer;
	END_VAR
END_METHOD


	(* Sets the canny edge detection thresholds. *)
	METHOD SetCannyThreshold : HRESULT
	VAR_INPUT
		(* Low threshold (> 0) *)
		nLow : DINT;
		(* High threshold (> nLow, usually 2 to 3 * nLow) *)
		nHigh : DINT;
	END_VAR
END_METHOD


	(* Sets the inverted ratio of the accumulator size in relation to the source image's size (e.g. a value of 2 means that the size is halved in both directions.) *)
	METHOD SetInvAccuRatio : HRESULT
	VAR_INPUT
		(* Inverted accumulator ratio (> 0) *)
		fInvAccuRatio : LREAL;
	END_VAR
END_METHOD


	(* Sets the number of R-table levels. *)
	METHOD SetLevels : HRESULT
	VAR_INPUT
		(* Number of R-table levels (> 0) *)
		nLevels : DINT;
	END_VAR
END_METHOD


	(* Sets the minimum distance between the centers of different objects. *)
	METHOD SetMinDist : HRESULT
	VAR_INPUT
		(* Minimum distance (> 0) *)
		fMinDist : LREAL;
	END_VAR
END_METHOD


	(* Sets the template image to search for in the Detect method. *)
	METHOD SetTemplate : HRESULT
	VAR_INPUT
		(* Template image (1 channel, USINT) *)
 {attribute 'GUID' := '70D42C6D-6F4E-4719-8B29-2883D5D59B1C'}
				ipImage : ITcVnImage;
	END_VAR
END_METHOD


	(* Sets the accumulator threshold, i.e. the number of votes required to detect a match (too small values lead to false detections). *)
	METHOD SetVotesThreshold : HRESULT
	VAR_INPUT
		(* Number of votes required to detect a match (> 0) *)
		nVotes : DINT;
	END_VAR
END_METHOD

END_FUNCTION_BLOCK

// Functions/Control Functions/F_VN_StartAbsWatchdog

	{attribute 'TcIecLibraryType'}
	{attribute 'external_name' := 'F_VN_StartAbsWatchdog_GUID_2A71E05D_731B_3642_11E7_B56A83924DB8'}
	(* Starts a cooperative watchdog given an absolute stop time. *)
	FUNCTION F_VN_StartAbsWatchdog : HRESULT
	VAR_INPUT
		tStop	:	DINT;	(* Stop time in us *)
		hrPrev	:	HRESULT;	(* HRESULT indicating the result of previous operations (If SUCCEEDED(hrPrev) equals false, no operation is executed.) *)
	END_VAR

END_FUNCTION

// Functions/Control Functions/F_VN_StartAbsWatchdogExp

	{attribute 'TcIecLibraryType'}
	{attribute 'external_name' := 'F_VN_StartAbsWatchdogExp_GUID_BA3B1008_3452_3AD6_3C52_2B3C9124286E'}
	(* Start a cooperative watchdog given an absolute stop time. (expert function) *)
	FUNCTION F_VN_StartAbsWatchdogExp : HRESULT
	VAR_INPUT
		tStop	:	DINT;	(* Stop time in us *)
		eWatchdogAccType	:	ETcWatchdogAccumulationType;	(* Accumalation method used for combining the results of multiple functions enclosed by this watchdog *)
		hrPrev	:	HRESULT;	(* HRESULT indicating the result of previous operations (If SUCCEEDED(hrPrev) equals false, no operation is executed.) *)
	END_VAR

END_FUNCTION

// Functions/Control Functions/F_VN_StartRelWatchdog

	{attribute 'TcIecLibraryType'}
	{attribute 'external_name' := 'F_VN_StartRelWatchdog_GUID_D1F2FBC4_412B_3812_367E_F558492366F7'}
	(* Starts a cooperative watchdog given a stop time relative to the current time. *)
	FUNCTION F_VN_StartRelWatchdog : HRESULT
	VAR_INPUT
		tStop	:	DINT;	(* Stop time in us *)
		hrPrev	:	HRESULT;	(* HRESULT indicating the result of previous operations (If SUCCEEDED(hrPrev) equals false, no operation is executed.) *)
	END_VAR

END_FUNCTION

// Functions/Control Functions/F_VN_StartRelWatchdogExp

	{attribute 'TcIecLibraryType'}
	{attribute 'external_name' := 'F_VN_StartRelWatchdogExp_GUID_D2B236B2_C38D_3222_13D1_71D34C52BEEE'}
	(* Start a cooperative watchdog given a stop time relative to the current time. (expert function) *)
	FUNCTION F_VN_StartRelWatchdogExp : HRESULT
	VAR_INPUT
		tStop	:	DINT;	(* Stop time in us *)
		eWatchdogAccType	:	ETcWatchdogAccumulationType;	(* Accumalation method used for combining the results of multiple functions enclosed by this watchdog *)
		hrPrev	:	HRESULT;	(* HRESULT indicating the result of previous operations (If SUCCEEDED(hrPrev) equals false, no operation is executed.) *)
	END_VAR

END_FUNCTION

// Functions/Control Functions/F_VN_StopWatchdog

	{attribute 'TcIecLibraryType'}
	{attribute 'external_name' := 'F_VN_StopWatchdog_GUID_B82A9514_2FB0_39A3_2A3D_67366D717D7D'}
	(* Stops a watchdog and provide runtime information. *)
	FUNCTION F_VN_StopWatchdog : HRESULT
	VAR_INPUT
		hrStartWatchdog	:	HRESULT;	(* HRESULT indicating the result of the function used to start the watchdog (If SUCCEEDED(hrStartWatchdog) equals false, no operation is executed.) *)
	END_VAR
	VAR_OUTPUT
		nFunctionsMonitored	:	ULINT;	(* Returns the number of functions monitored *)
		nFractionProcessed	:	UDINT;	(* Returns the fraction processed accumulated over the monitored functions in percent *)
		tRest	:	DINT;	(* Returns the remaining computation time in us (may be negative) *)
	END_VAR

END_FUNCTION

// Functions/Image Segmentation/F_VN_AdaptiveThreshold

	{attribute 'TcIecLibraryType'}
	{attribute 'external_name' := 'F_VN_AdaptiveThreshold_GUID_567ECDBF_A4C8_308E_252D_4E80DB2717E4'}
	(* Apply an adaptive threshold to a gray level image. *)
	FUNCTION F_VN_AdaptiveThreshold : HRESULT
	VAR_INPUT
		ipSrcImage	:	ITcVnImage;	(* Source image (1 channel, elements of type USINT) *)
		ipDestImage	:	REFERENCE TO ITcVnImage;	(* Destination image (An appropriate destination image will be created if required.) *)
		fMaxValue	:	LREAL;	(* Value assigned to pixels for which the threshold condition is true *)
		hrPrev	:	HRESULT;	(* HRESULT indicating the result of previous operations (If SUCCEEDED(hrPrev) equals false, no operation is executed.) *)
	END_VAR

END_FUNCTION

// Functions/Image Segmentation/F_VN_AdaptiveThresholdExp

	{attribute 'TcIecLibraryType'}
	{attribute 'external_name' := 'F_VN_AdaptiveThresholdExp_GUID_03DC4893_5B25_3488_221F_ED5AECEC24C0'}
	(* Apply an adaptive threshold to a gray level image. (expert function) *)
	FUNCTION F_VN_AdaptiveThresholdExp : HRESULT
	VAR_INPUT
		ipSrcImage	:	ITcVnImage;	(* Source image (1 channel, elements of type USINT) *)
		ipDestImage	:	REFERENCE TO ITcVnImage;	(* Destination image (An appropriate destination image will be created if required.) *)
		fMaxValue	:	LREAL;	(* Value assigned to pixels for which the threshold condition is true *)
		eAdaptiveMethod	:	ETcVnAdaptiveThresholdMethod;	(* Adaptive threshold method to be applied (MEAN: threshold value will be calculated as a mean of the nBlockSize x nBlockSize neighborhood of (x,y) minus fConstant. GAUSSIAN: threshold value is a weighted sum (cross-correlation with a Gaussian window) of the nBlockSize x nBlockSize neighborhood of (x,y) minus fConstant. *)
		eThresholdType	:	ETcVnThresholdType;	(* Threshold type to be applied (only BINARY and BINARY_INV are supported) *)
		nBlockSize	:	UDINT;	(* Size of the pixel neighborhood to calculate the local threshold (3, 5, 7, ...) *)
		fConstant	:	LREAL;	(* Constant that is subtracted from the weighted mean of the pixel neighborhood, which leads to the local threshold *)
		hrPrev	:	HRESULT;	(* HRESULT indicating the result of previous operations (If SUCCEEDED(hrPrev) equals false, no operation is executed.) *)
	END_VAR

END_FUNCTION

// Functions/Image Segmentation/F_VN_CheckColorRange

	{attribute 'TcIecLibraryType'}
	{attribute 'external_name' := 'F_VN_CheckColorRange_GUID_B8C720DA_1F7F_3A23_3608_487A19EE46AC'}
	(* Check if the pixel values of an image lie in a given range. The destination image has the same size as the source image but only one channel with
          a pixel element size of 8 bit. Its elements are set to 255 if the corresponding pixels of the source image are in the checked range and set to 0 otherwise. *)
	FUNCTION F_VN_CheckColorRange : HRESULT
	VAR_INPUT
		ipSrcImage	:	ITcVnImage;	(* Source image *)
		ipDestImage	:	REFERENCE TO ITcVnImage;	(* Destination image (An appropriate destination image will be created if required.) *)
		aLowerBounds	:	REFERENCE TO TcVnVector4_LREAL;	(* Channel-wise lower bounds (Unused channels are ignored.) *)
		aUpperBounds	:	REFERENCE TO TcVnVector4_LREAL;	(* Channel-wise upper bounds (Unused channels are ignored.) *)
		hrPrev	:	HRESULT;	(* HRESULT indicating the result of previous operations (If SUCCEEDED(hrPrev) equals false, no operation is executed.) *)
	END_VAR

END_FUNCTION

// Functions/Image Segmentation/F_VN_Threshold

	{attribute 'TcIecLibraryType'}
	{attribute 'external_name' := 'F_VN_Threshold_GUID_137D3CD0_456D_3B2E_122F_E3D0A8D69801'}
	(* Apply a fixed threshold or a dynamic threshold according to Otsu. *)
	FUNCTION F_VN_Threshold : HRESULT
	VAR_INPUT
		ipSrcImage	:	ITcVnImage;	(* Source image (For Otsu and Triangle threshold types, only 1 channel of TCVN_ET_USINT is supported) *)
		ipDestImage	:	REFERENCE TO ITcVnImage;	(* Destination image (An appropriate destination image will be created if required.) *)
		fThreshold	:	LREAL;	(* Fixed threshold (unused if dynamic thresholding is selected) *)
		fMaxValue	:	LREAL;	(* Maximum pixel value *)
		eThresholdType	:	ETcVnThresholdType;	(* Threshold type to be applied *)
		hrPrev	:	HRESULT;	(* HRESULT indicating the result of previous operations (If SUCCEEDED(hrPrev) equals false, no operation is executed.) *)
	END_VAR

END_FUNCTION

// Functions/Image Segmentation/F_VN_WatershedSegmentationExp

	{attribute 'TcIecLibraryType'}
	{attribute 'external_name' := 'F_VN_WatershedSegmentationExp_GUID_E286F9D3_CBD4_3005_1C99_0EF8D9099032'}
	(* Apply a marker-based watershed segmentation. (expert function) *)
	FUNCTION F_VN_WatershedSegmentationExp : HRESULT
	VAR_INPUT
		ipSrcImage	:	ITcVnImage;	(* Source image (USINT, 3 channels) *)
		ipDestImage	:	REFERENCE TO ITcVnImage;	(* Destination image (DINT, 1 channel. An appropriate image will be created if required.) *)
		ipMarkers	:	ITcVnImage;	(* Marker image (DINT, 1 channel) *)
		hrPrev	:	HRESULT;	(* HRESULT indicating the result of previous operations (If SUCCEEDED(hrPrev) equals false, no operation is executed.) *)
	END_VAR

END_FUNCTION

// Functions/Algebraic Container Operations/F_VN_AddContainers

	{attribute 'TcIecLibraryType'}
	{attribute 'external_name' := 'F_VN_AddContainers_GUID_D30AD915_864D_3B82_2778_D82BFD50BA88'}
	(* Element-wise addition of two containers (same length and type). *)
	FUNCTION F_VN_AddContainers : HRESULT
	VAR_INPUT
		ipSrcContainer1	:	ITcVnContainer;	(* Source container 1 *)
		ipSrcContainer2	:	ITcVnContainer;	(* Source container 2 *)
		ipDestContainer	:	REFERENCE TO ITcVnContainer;	(* Returns the resulting container *)
		hrPrev	:	HRESULT;	(* HRESULT indicating the result of previous operations (If SUCCEEDED(hrPrev) equals false, no operation is executed.) *)
	END_VAR

END_FUNCTION

// Functions/Algebraic Container Operations/F_VN_BitwiseAndContainers

	{attribute 'TcIecLibraryType'}
	{attribute 'external_name' := 'F_VN_BitwiseAndContainers_GUID_0CB7C0DF_A0ED_3B5C_36DD_0E8AA14E9BB4'}
	(* Element-wise application of a bit-wise AND operator to two containers (same length and type, integer only). *)
	FUNCTION F_VN_BitwiseAndContainers : HRESULT
	VAR_INPUT
		ipSrcContainer1	:	ITcVnContainer;	(* Source container 1 *)
		ipSrcContainer2	:	ITcVnContainer;	(* Source container 2 *)
		ipDestContainer	:	REFERENCE TO ITcVnContainer;	(* Returns the resulting container *)
		hrPrev	:	HRESULT;	(* HRESULT indicating the result of previous operations (If SUCCEEDED(hrPrev) equals false, no operation is executed.) *)
	END_VAR

END_FUNCTION

// Functions/Algebraic Container Operations/F_VN_BitwiseNotContainer

	{attribute 'TcIecLibraryType'}
	{attribute 'external_name' := 'F_VN_BitwiseNotContainer_GUID_10D6DB3B_69E8_336F_310A_DA9C24871695'}
	(* Element-wise application of a bit-wise NOT operator to a container (integer only). *)
	FUNCTION F_VN_BitwiseNotContainer : HRESULT
	VAR_INPUT
		ipSrcContainer	:	ITcVnContainer;	(* Source container *)
		ipDestContainer	:	REFERENCE TO ITcVnContainer;	(* Returns the resulting container *)
		hrPrev	:	HRESULT;	(* HRESULT indicating the result of previous operations (If SUCCEEDED(hrPrev) equals false, no operation is executed.) *)
	END_VAR

END_FUNCTION

// Functions/Algebraic Container Operations/F_VN_BitwiseOrContainers

	{attribute 'TcIecLibraryType'}
	{attribute 'external_name' := 'F_VN_BitwiseOrContainers_GUID_17B141E3_C244_33E8_2160_EE54A47B1366'}
	(* Element-wise application of a bit-wise OR operator to two containers (same length and type, integer only). *)
	FUNCTION F_VN_BitwiseOrContainers : HRESULT
	VAR_INPUT
		ipSrcContainer1	:	ITcVnContainer;	(* Source container 1 *)
		ipSrcContainer2	:	ITcVnContainer;	(* Source container 2 *)
		ipDestContainer	:	REFERENCE TO ITcVnContainer;	(* Returns the resulting container *)
		hrPrev	:	HRESULT;	(* HRESULT indicating the result of previous operations (If SUCCEEDED(hrPrev) equals false, no operation is executed.) *)
	END_VAR

END_FUNCTION

// Functions/Algebraic Container Operations/F_VN_BitwiseXorContainers

	{attribute 'TcIecLibraryType'}
	{attribute 'external_name' := 'F_VN_BitwiseXorContainers_GUID_57C8BF82_AC91_3626_3BDD_CF193908D1BE'}
	(* Element-wise application of a bit-wise XOR operator to two containers (same length and type, integer only). *)
	FUNCTION F_VN_BitwiseXorContainers : HRESULT
	VAR_INPUT
		ipSrcContainer1	:	ITcVnContainer;	(* Source container 1 *)
		ipSrcContainer2	:	ITcVnContainer;	(* Source container 2 *)
		ipDestContainer	:	REFERENCE TO ITcVnContainer;	(* Returns the resulting container *)
		hrPrev	:	HRESULT;	(* HRESULT indicating the result of previous operations (If SUCCEEDED(hrPrev) equals false, no operation is executed.) *)
	END_VAR

END_FUNCTION

// Functions/Algebraic Container Operations/F_VN_DivideContainers

	{attribute 'TcIecLibraryType'}
	{attribute 'external_name' := 'F_VN_DivideContainers_GUID_A8B84557_0081_394E_2C60_F5DB05D388E5'}
	(* Element-wise division of two containers (same length and type). In case of integer division by zero, the resulting element is set to 0 and S_DIVISION_BY_ZERO is returned instead of S_OK (value can be changed in F_VN_DivideContainersExp). *)
	FUNCTION F_VN_DivideContainers : HRESULT
	VAR_INPUT
		ipSrcContainer1	:	ITcVnContainer;	(* Source container 1 *)
		ipSrcContainer2	:	ITcVnContainer;	(* Source container 2 *)
		ipDestContainer	:	REFERENCE TO ITcVnContainer;	(* Returns the resulting container *)
		hrPrev	:	HRESULT;	(* HRESULT indicating the result of previous operations (If SUCCEEDED(hrPrev) equals false, no operation is executed.) *)
	END_VAR

END_FUNCTION

// Functions/Algebraic Container Operations/F_VN_DivideContainersExp

	{attribute 'TcIecLibraryType'}
	{attribute 'external_name' := 'F_VN_DivideContainersExp_GUID_B0A58345_C222_376C_1405_49F4221D3DA8'}
	(* Element-wise division of two containers (same length and type). In case of integer division by zero, the resulting element is set to nIntDivideByZeroResult and S_DIVISION_BY_ZERO is returned instead of S_OK. (expert function) *)
	FUNCTION F_VN_DivideContainersExp : HRESULT
	VAR_INPUT
		ipSrcContainer1	:	ITcVnContainer;	(* Source container 1 *)
		ipSrcContainer2	:	ITcVnContainer;	(* Source container 2 *)
		ipDestContainer	:	REFERENCE TO ITcVnContainer;	(* Returns the resulting container *)
		nIntDivideByZeroResult	:	LINT;	(* Value set as result in case of integer division by zero *)
		hrPrev	:	HRESULT;	(* HRESULT indicating the result of previous operations (If SUCCEEDED(hrPrev) equals false, no operation is executed.) *)
	END_VAR

END_FUNCTION

// Functions/Algebraic Container Operations/F_VN_MaxContainer

	{attribute 'TcIecLibraryType'}
	{attribute 'external_name' := 'F_VN_MaxContainer_GUID_60252BE8_1CD2_3505_2D79_2364B3A7914F'}
	(* Element-wise maximum of two containers (same length and type). *)
	FUNCTION F_VN_MaxContainer : HRESULT
	VAR_INPUT
		ipSrcContainer1	:	ITcVnContainer;	(* Source container 1 *)
		ipSrcContainer2	:	ITcVnContainer;	(* Source container 2 *)
		ipDestContainer	:	REFERENCE TO ITcVnContainer;	(* Returns the resulting container *)
		hrPrev	:	HRESULT;	(* HRESULT indicating the result of previous operations (If SUCCEEDED(hrPrev) equals false, no operation is executed.) *)
	END_VAR

END_FUNCTION

// Functions/Algebraic Container Operations/F_VN_MinContainer

	{attribute 'TcIecLibraryType'}
	{attribute 'external_name' := 'F_VN_MinContainer_GUID_EA44B26A_F97A_3365_16BB_087569331F7B'}
	(* Element-wise minimum of two containers (same length and type). *)
	FUNCTION F_VN_MinContainer : HRESULT
	VAR_INPUT
		ipSrcContainer1	:	ITcVnContainer;	(* Source container 1 *)
		ipSrcContainer2	:	ITcVnContainer;	(* Source container 2 *)
		ipDestContainer	:	REFERENCE TO ITcVnContainer;	(* Returns the resulting container *)
		hrPrev	:	HRESULT;	(* HRESULT indicating the result of previous operations (If SUCCEEDED(hrPrev) equals false, no operation is executed.) *)
	END_VAR

END_FUNCTION

// Functions/Algebraic Container Operations/F_VN_MultiplyContainers

	{attribute 'TcIecLibraryType'}
	{attribute 'external_name' := 'F_VN_MultiplyContainers_GUID_F2FEADE1_7C5F_37A1_2C23_01A0A229AADE'}
	(* Element-wise multiplication of two containers (same length and type). *)
	FUNCTION F_VN_MultiplyContainers : HRESULT
	VAR_INPUT
		ipSrcContainer1	:	ITcVnContainer;	(* Source container 1 *)
		ipSrcContainer2	:	ITcVnContainer;	(* Source container 2 *)
		ipDestContainer	:	REFERENCE TO ITcVnContainer;	(* Returns the resulting container *)
		hrPrev	:	HRESULT;	(* HRESULT indicating the result of previous operations (If SUCCEEDED(hrPrev) equals false, no operation is executed.) *)
	END_VAR

END_FUNCTION

